Universal Robots PolyScope program: DAS428_958_02_MAR_21_DAS_lado_derecho.urp

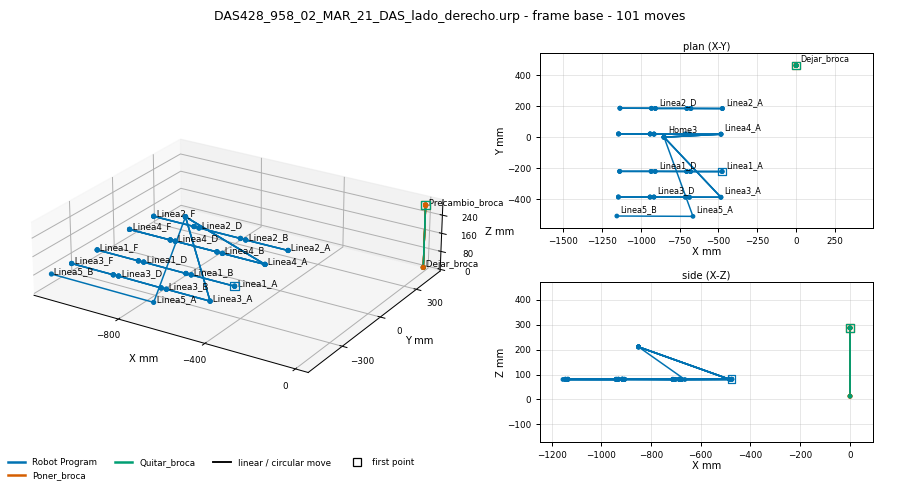
[picture p0: tool path of DAS428_958_02_MAR_21_DAS_lado_derecho.urp in frame base, 101 of 219 moves have a stored position in this frame; points joined in program order, loops and branches not executed]
Program DAS428_958_02_MAR_21_DAS_lado_derecho (installation=instalacion_26_FEB_21 directory=/programs/derecho createdIn=5.6.0.90886 lastSavedIn=5.6.0.90886 robotSerialNumber=20195001785)
Calibrated DH parameters: a=[0.000107, -0.568984, -0.552934, -0.00001, -0.000063, 0]; d=[0.180718, -257.998067, 200.685024, 57.48776, 0.119923, 0.115353]; alpha=[1.571119, 0.000876, -0.002498, 1.571178, -1.570523, 0]; deltaTheta=[0, -0.378191, 0.631587, -0.253396, 0, 0]
Robot Program (runOnlyOnce=false)
  Folder Variables
    bajada_broca := p[0,0,-0.008,0,0,0]
    barrenos_menos1 := 0
    barreno_actual := 0
    posicion := p[0,0,300,0,0,0]
    cambiar_broca := False
    barrenos_hechos := 0
    eje7 := 0
    Wait Sleep waitTime=0.5
  Folder Home
    Wait Sleep waitTime=0.3
    SafeHome (positionOptionType=SPEED_AND_ACCELERATION speed=1.047198 acceleration=1.396263 nextMotionTime=2)
    SuppressedNode
      MoveL speed 250 mm/s, acceleration 1200 mm/s^2 (useActiveTCP=true) feature=Base
        Waypoint home_trans: TCP in base x=-171.077 y=546.65 z=109.574 mm, rx=0.1544 ry=3.1247 rz=-0.2011 rad; joints [-91.802, -93.053, 127.954, -27.005, -275.278, -0.192] deg; TCP offset x=0.411 y=-218.298 z=37.994 mm, rx=1.558 ry=-0.1255 rz=0.1212 rad
    Wait Sleep waitTime=0.3
    iniciando_prog := True
    Call Poner_broca
  Folder Posicion2
    eje7 := 2
    Folder Broca_1
      Folder Linea1
        Folder Marcar_puntos
          MoveL speed 100 mm/s, acceleration 500 mm/s^2 (useActiveTCP=true) feature=Base
            SafeHome (positionOptionType=SPEED_AND_ACCELERATION speed=1.047198 acceleration=1.396263 nextMotionTime=2)
            Waypoint Linea1_A: TCP in base x=-476.23 y=-221.4 z=80.998 mm, rx=2.0263 ry=-2.3929 rz=-0.0208 rad; joints [8.239, -98.147, 138.323, -40.444, -261.448, -0.264] deg; TCP offset x=0.411 y=-218.298 z=37.994 mm, rx=1.558 ry=-0.1255 rz=0.1212 rad
            Waypoint Linea1_B: TCP in base x=-679.349 y=-221.301 z=80.412 mm, rx=2.0263 ry=-2.3929 rz=-0.0208 rad; joints [5.2, -80.225, 120.117, -40.154, -264.492, -0.236] deg
            Waypoint Linea1_C: TCP in base x=-704.534 y=-220.853 z=80.143 mm, rx=2.0263 ry=-2.3929 rz=-0.0208 rad; joints [4.927, -78.214, 117.618, -39.664, -264.765, -0.234] deg
            Waypoint Linea1_D: TCP in base x=-907.519 y=-220.332 z=80.645 mm, rx=2.0263 ry=-2.3929 rz=-0.0208 rad; joints [3.596, -62.527, 94.913, -32.645, -266.086, -0.228] deg
            Waypoint Linea1_E: TCP in base x=-933.182 y=-220.332 z=80.091 mm, rx=2.0263 ry=-2.3929 rz=-0.0208 rad; joints [3.48, -60.486, 91.71, -31.482, -266.199, -0.227] deg
            Waypoint Linea1_F: TCP in base x=-1136.071 y=-220.201 z=80.22 mm, rx=2.0263 ry=-2.3929 rz=-0.0208 rad; joints [2.763, -42.904, 61.27, -18.625, -266.887, -0.23] deg
        Folder AB
          'desbaste_inicial'
          bajada_broca := p[0,0,-0.008,0,0,0]
          barrenos_menos1 := 8
          barreno_actual := 0
          Loop While (checkContinuously=false) expression=barreno_actual≤barrenos_menos1
            Folder Perforacion
              MoveL speed 100 mm/s, acceleration 500 mm/s^2 (useActiveTCP=true) feature=Base
                internos := interpolate_pose(Linea1_A, Linea1_B, barreno_actual/barrenos_menos1)
                Waypoint Waypoint (Variable): variable=internos
                'desbaste_inicial'
                bajada_broca := p[0,0,-0.008,0,0,0]
                bajada := p[0,0,0.008,0,0,0]
                MoveDirectionNode (selectedDirection=ZMinus toolParams=0.003, 0.005)
                  Until DISTANCE (allowActions=false deceleration=3 distanceNodeType=STOP) Distance=0.045; motionParameters(blendRadius=0)
                Popup Message (haltProgram=false message=punto contacto alanzdo inputType=Text)
                MoveDirectionNode (selectedDirection=ZPlus toolParams=0.003, 0.005)
                  Until DISTANCE (allowActions=false deceleration=3 distanceNodeType=STOP) Distance=0.002; motionParameters(blendRadius=0)
                Wait Sleep waitTime=0.3
                Set DigitalOutput pin=config_out[1]; digitalValue=1
                Wait Sleep waitTime=0.3
                Loop Counting (count=3) loopVariable(name=Loop_11)
                  bajar := pose_add(get_actual_tcp_pose(), bajada_broca)
                  Waypoint Waypoint (Variable): motionParameters(jointSpeed=1.047198 jointAcceleration=1.396263 cartesianSpeed=0.001 cartesianAcceleration=0.005); variable=bajar
                  subir := pose_sub(get_actual_tcp_pose(), bajada_broca)
                  Waypoint Waypoint (Variable): motionParameters(jointSpeed=1.047198 jointAcceleration=1.396263 cartesianSpeed=0.005 cartesianAcceleration=0.01); variable=subir
                  bajada_broca := pose_sub(bajada_broca, bajada)
                MoveDirectionNode (selectedDirection=ZPlus toolParams=0.03, 0.035)
                  Until DISTANCE (allowActions=false deceleration=3 distanceNodeType=STOP) Distance=0.06; motionParameters(blendRadius=0)
                Set DigitalOutput pin=config_out[1]; digitalValue=0
                barreno_actual := barreno_actual+1
                Call Quitar_broca
                Call Poner_broca
        Folder CD
          'desbaste_inicial'
          bajada_broca := p[0,0,-0.008,0,0,0]
          barrenos_menos1 := 8
          barreno_actual := 0
          Loop While (checkContinuously=false) expression=barreno_actual≤barrenos_menos1
            Folder Perforacion
              MoveL speed 100 mm/s, acceleration 500 mm/s^2 (useActiveTCP=true) feature=Base
                internos := interpolate_pose(Linea1_C, Linea1_D, barreno_actual/barrenos_menos1)
                Waypoint Waypoint (Variable): variable=internos
                'desbaste_inicial'
                bajada_broca := p[0,0,-0.008,0,0,0]
                bajada := p[0,0,0.008,0,0,0]
                MoveDirectionNode (selectedDirection=ZMinus toolParams=0.003, 0.005)
                  Until DISTANCE (allowActions=false deceleration=3 distanceNodeType=STOP) Distance=0.045; motionParameters(blendRadius=0)
                Popup Message (haltProgram=false message=punto contacto alanzdo inputType=Text)
                MoveDirectionNode (selectedDirection=ZPlus toolParams=0.003, 0.005)
                  Until DISTANCE (allowActions=false deceleration=3 distanceNodeType=STOP) Distance=0.002; motionParameters(blendRadius=0)
                Wait Sleep waitTime=0.3
                Set DigitalOutput pin=config_out[1]; digitalValue=1
                Wait Sleep waitTime=0.3
                Loop Counting (count=3) loopVariable(name=Loop_14)
                  bajar := pose_add(get_actual_tcp_pose(), bajada_broca)
                  Waypoint Waypoint (Variable): motionParameters(jointSpeed=1.047198 jointAcceleration=1.396263 cartesianSpeed=0.001 cartesianAcceleration=0.005); variable=bajar
                  subir := pose_sub(get_actual_tcp_pose(), bajada_broca)
                  Waypoint Waypoint (Variable): motionParameters(jointSpeed=1.047198 jointAcceleration=1.396263 cartesianSpeed=0.005 cartesianAcceleration=0.01); variable=subir
                  bajada_broca := pose_sub(bajada_broca, bajada)
                MoveDirectionNode (selectedDirection=ZPlus toolParams=0.03, 0.035)
                  Until DISTANCE (allowActions=false deceleration=3 distanceNodeType=STOP) Distance=0.06; motionParameters(blendRadius=0)
                Set DigitalOutput pin=config_out[1]; digitalValue=0
                barreno_actual := barreno_actual+1
                Call Quitar_broca
                Call Poner_broca
        Folder EF
          'desbaste_inicial'
          bajada_broca := p[0,0,-0.008,0,0,0]
          barrenos_menos1 := 8
          barreno_actual := 0
          Loop While (checkContinuously=false) expression=barreno_actual≤barrenos_menos1
            Folder Perforacion
              MoveL speed 100 mm/s, acceleration 500 mm/s^2 (useActiveTCP=true) feature=Base
                internos := interpolate_pose(Linea1_E, Linea1_F, barreno_actual/barrenos_menos1)
                Waypoint Waypoint (Variable): variable=internos
                'desbaste_inicial'
                bajada_broca := p[0,0,-0.008,0,0,0]
                bajada := p[0,0,0.008,0,0,0]
                MoveDirectionNode (selectedDirection=ZMinus toolParams=0.003, 0.005)
                  Until DISTANCE (allowActions=false deceleration=3 distanceNodeType=STOP) Distance=0.045; motionParameters(blendRadius=0)
                Popup Message (haltProgram=false message=punto contacto alanzdo inputType=Text)
                MoveDirectionNode (selectedDirection=ZPlus toolParams=0.003, 0.005)
                  Until DISTANCE (allowActions=false deceleration=3 distanceNodeType=STOP) Distance=0.002; motionParameters(blendRadius=0)
                Wait Sleep waitTime=0.3
                Set DigitalOutput pin=config_out[1]; digitalValue=1
                Wait Sleep waitTime=0.3
                Loop Counting (count=3) loopVariable(name=Loop_16)
                  bajar := pose_add(get_actual_tcp_pose(), bajada_broca)
                  Waypoint Waypoint (Variable): motionParameters(jointSpeed=1.047198 jointAcceleration=1.396263 cartesianSpeed=0.001 cartesianAcceleration=0.005); variable=bajar
                  subir := pose_sub(get_actual_tcp_pose(), bajada_broca)
                  Waypoint Waypoint (Variable): motionParameters(jointSpeed=1.047198 jointAcceleration=1.396263 cartesianSpeed=0.005 cartesianAcceleration=0.01); variable=subir
                  bajada_broca := pose_sub(bajada_broca, bajada)
                MoveDirectionNode (selectedDirection=ZPlus toolParams=0.03, 0.035)
                  Until DISTANCE (allowActions=false deceleration=3 distanceNodeType=STOP) Distance=0.06; motionParameters(blendRadius=0)
                Set DigitalOutput pin=config_out[1]; digitalValue=0
                barreno_actual := barreno_actual+1
                Call Quitar_broca
                Call Poner_broca
      Popup Message (haltProgram=false message=Linea1 con chica Terminada! inputType=Text)
      Folder Linea2
        Folder Marcar_puntos
          MoveL speed 100 mm/s, acceleration 500 mm/s^2 (useActiveTCP=true) feature=Base
            Waypoint Linea2_A: TCP in base x=-474.583 y=184.454 z=81.011 mm, rx=2.0263 ry=-2.3928 rz=-0.0209 rad; joints [-57.964, -100.998, 140.513, -39.882, -327.65, 0.115] deg; TCP offset x=0.411 y=-218.298 z=37.994 mm, rx=1.558 ry=-0.1255 rz=0.1212 rad
            Waypoint Linea2_B: TCP in base x=-677.479 y=185.069 z=80.034 mm, rx=2.0263 ry=-2.3928 rz=-0.0209 rad; joints [-37.655, -81.603, 121.85, -40.529, -307.349, -0.029] deg
            Waypoint Linea2_C: TCP in base x=-703.112 y=185.207 z=80.706 mm, rx=2.0263 ry=-2.3928 rz=-0.0209 rad; joints [-36.031, -79.522, 119.204, -39.96, -305.725, -0.038] deg
            Waypoint Linea2_D: TCP in base x=-906.15 y=185.294 z=81.03 mm, rx=2.0263 ry=-2.3928 rz=-0.0209 rad; joints [-26.739, -63.46, 96.339, -33.14, -296.423, -0.088] deg
            Waypoint Linea2_E: TCP in base x=-931.212 y=185.988 z=81.375 mm, rx=2.0263 ry=-2.3928 rz=-0.0209 rad; joints [-25.954, -61.479, 93.157, -31.938, -295.635, -0.093] deg
            Waypoint Linea2_F: TCP in base x=-1134.161 y=186.61 z=81.262 mm, rx=2.0263 ry=-2.3928 rz=-0.0209 rad; joints [-20.753, -43.887, 62.952, -19.317, -290.406, -0.124] deg
        Folder AB
          'desbaste_inicial'
          bajada_broca := p[0,0,-0.008,0,0,0]
          barrenos_menos1 := 8
          barreno_actual := 0
          Loop While (checkContinuously=false) expression=barreno_actual≤barrenos_menos1
            Folder Perforacion
              MoveL speed 100 mm/s, acceleration 500 mm/s^2 (useActiveTCP=true) feature=Base
                internos := interpolate_pose(Linea2_A, Linea2_B, barreno_actual/barrenos_menos1)
                Waypoint Waypoint (Variable): variable=internos
                'desbaste_inicial'
                bajada_broca := p[0,0,-0.008,0,0,0]
                bajada := p[0,0,0.008,0,0,0]
                MoveDirectionNode (selectedDirection=ZMinus toolParams=0.003, 0.005)
                  Until DISTANCE (allowActions=false deceleration=3 distanceNodeType=STOP) Distance=0.045; motionParameters(blendRadius=0)
                Popup Message (haltProgram=false message=punto contacto alanzdo inputType=Text)
                MoveDirectionNode (selectedDirection=ZPlus toolParams=0.003, 0.005)
                  Until DISTANCE (allowActions=false deceleration=3 distanceNodeType=STOP) Distance=0.002; motionParameters(blendRadius=0)
                Wait Sleep waitTime=0.3
                Set DigitalOutput pin=config_out[1]; digitalValue=1
                Wait Sleep waitTime=0.3
                Loop Counting (count=3) loopVariable(name=Loop_2)
                  bajar := pose_add(get_actual_tcp_pose(), bajada_broca)
                  Waypoint Waypoint (Variable): motionParameters(jointSpeed=1.047198 jointAcceleration=1.396263 cartesianSpeed=0.001 cartesianAcceleration=0.005); variable=bajar
                  subir := pose_sub(get_actual_tcp_pose(), bajada_broca)
                  Waypoint Waypoint (Variable): motionParameters(jointSpeed=1.047198 jointAcceleration=1.396263 cartesianSpeed=0.005 cartesianAcceleration=0.01); variable=subir
                  bajada_broca := pose_sub(bajada_broca, bajada)
                MoveDirectionNode (selectedDirection=ZPlus toolParams=0.03, 0.035)
                  Until DISTANCE (allowActions=false deceleration=3 distanceNodeType=STOP) Distance=0.06; motionParameters(blendRadius=0)
                Set DigitalOutput pin=config_out[1]; digitalValue=0
                barreno_actual := barreno_actual+1
                Call Quitar_broca
                Call Poner_broca
        Folder CD
          'desbaste_inicial'
          bajada_broca := p[0,0,-0.008,0,0,0]
          barrenos_menos1 := 8
          barreno_actual := 0
          Loop While (checkContinuously=false) expression=barreno_actual≤barrenos_menos1
            Folder Perforacion
              MoveL speed 100 mm/s, acceleration 500 mm/s^2 (useActiveTCP=true) feature=Base
                internos := interpolate_pose(Linea2_C, Linea2_D, barreno_actual/barrenos_menos1)
                Waypoint Waypoint (Variable): variable=internos
                'desbaste_inicial'
                bajada_broca := p[0,0,-0.008,0,0,0]
                bajada := p[0,0,0.008,0,0,0]
                MoveDirectionNode (selectedDirection=ZMinus toolParams=0.003, 0.005)
                  Until DISTANCE (allowActions=false deceleration=3 distanceNodeType=STOP) Distance=0.045; motionParameters(blendRadius=0)
                Popup Message (haltProgram=false message=punto contacto alanzdo inputType=Text)
                MoveDirectionNode (selectedDirection=ZPlus toolParams=0.003, 0.005)
                  Until DISTANCE (allowActions=false deceleration=3 distanceNodeType=STOP) Distance=0.002; motionParameters(blendRadius=0)
                Wait Sleep waitTime=0.3
                Set DigitalOutput pin=config_out[1]; digitalValue=1
                Wait Sleep waitTime=0.3
                Loop Counting (count=3) loopVariable(name=Loop_5)
                  bajar := pose_add(get_actual_tcp_pose(), bajada_broca)
                  Waypoint Waypoint (Variable): motionParameters(jointSpeed=1.047198 jointAcceleration=1.396263 cartesianSpeed=0.001 cartesianAcceleration=0.005); variable=bajar
                  subir := pose_sub(get_actual_tcp_pose(), bajada_broca)
                  Waypoint Waypoint (Variable): motionParameters(jointSpeed=1.047198 jointAcceleration=1.396263 cartesianSpeed=0.005 cartesianAcceleration=0.01); variable=subir
                  bajada_broca := pose_sub(bajada_broca, bajada)
                MoveDirectionNode (selectedDirection=ZPlus toolParams=0.03, 0.035)
                  Until DISTANCE (allowActions=false deceleration=3 distanceNodeType=STOP) Distance=0.06; motionParameters(blendRadius=0)
                Set DigitalOutput pin=config_out[1]; digitalValue=0
                barreno_actual := barreno_actual+1
                Call Quitar_broca
                Call Poner_broca
        Folder EF
          'desbaste_inicial'
          bajada_broca := p[0,0,-0.008,0,0,0]
          barrenos_menos1 := 8
          barreno_actual := 0
          Loop While (checkContinuously=false) expression=barreno_actual≤barrenos_menos1
            Folder Perforacion
              MoveL speed 100 mm/s, acceleration 500 mm/s^2 (useActiveTCP=true) feature=Base
                internos := interpolate_pose(Linea2_E, Linea2_F, barreno_actual/barrenos_menos1)
                Waypoint Waypoint (Variable): variable=internos
                'desbaste_inicial'
                bajada_broca := p[0,0,-0.008,0,0,0]
                bajada := p[0,0,0.008,0,0,0]
                MoveDirectionNode (selectedDirection=ZMinus toolParams=0.003, 0.005)
                  Until DISTANCE (allowActions=false deceleration=3 distanceNodeType=STOP) Distance=0.045; motionParameters(blendRadius=0)
                Popup Message (haltProgram=false message=punto contacto alanzdo inputType=Text)
                MoveDirectionNode (selectedDirection=ZPlus toolParams=0.003, 0.005)
                  Until DISTANCE (allowActions=false deceleration=3 distanceNodeType=STOP) Distance=0.002; motionParameters(blendRadius=0)
                Wait Sleep waitTime=0.3
                Set DigitalOutput pin=config_out[1]; digitalValue=1
                Wait Sleep waitTime=0.3
                Loop Counting (count=3) loopVariable(name=Loop_9)
                  bajar := pose_add(get_actual_tcp_pose(), bajada_broca)
                  Waypoint Waypoint (Variable): motionParameters(jointSpeed=1.047198 jointAcceleration=1.396263 cartesianSpeed=0.001 cartesianAcceleration=0.005); variable=bajar
                  subir := pose_sub(get_actual_tcp_pose(), bajada_broca)
                  Waypoint Waypoint (Variable): motionParameters(jointSpeed=1.047198 jointAcceleration=1.396263 cartesianSpeed=0.005 cartesianAcceleration=0.01); variable=subir
                  bajada_broca := pose_sub(bajada_broca, bajada)
                MoveDirectionNode (selectedDirection=ZPlus toolParams=0.03, 0.035)
                  Until DISTANCE (allowActions=false deceleration=3 distanceNodeType=STOP) Distance=0.06; motionParameters(blendRadius=0)
                Set DigitalOutput pin=config_out[1]; digitalValue=0
                barreno_actual := barreno_actual+1
                If barreno_actual≥barrenos_menos1
                  cambiar_broca := True
                Call Quitar_broca
                Call Poner_broca
      Popup Message (haltProgram=false message=Linea2 con chica Terminada! inputType=Text)
    Folder Broca_2
      Folder Linea1
        Folder Marcar_puntos
          MoveL speed 100 mm/s, acceleration 500 mm/s^2 (useActiveTCP=true) feature=Base
            Waypoint Linea1_A: TCP in base x=-476.23 y=-221.4 z=80.998 mm, rx=2.0263 ry=-2.3929 rz=-0.0208 rad; joints [8.239, -98.147, 138.323, -40.444, -261.448, -0.264] deg; TCP offset x=0.411 y=-218.298 z=37.994 mm, rx=1.558 ry=-0.1255 rz=0.1212 rad
            Waypoint Linea1_B: TCP in base x=-679.349 y=-221.301 z=80.412 mm, rx=2.0263 ry=-2.3929 rz=-0.0208 rad; joints [5.2, -80.225, 120.117, -40.154, -264.492, -0.236] deg
            Waypoint Linea1_C: TCP in base x=-704.534 y=-220.853 z=80.143 mm, rx=2.0263 ry=-2.3929 rz=-0.0208 rad; joints [4.927, -78.214, 117.618, -39.664, -264.765, -0.234] deg
            Waypoint Linea1_D: TCP in base x=-907.519 y=-220.332 z=80.645 mm, rx=2.0263 ry=-2.3929 rz=-0.0208 rad; joints [3.596, -62.527, 94.913, -32.645, -266.086, -0.228] deg
            Waypoint Linea1_E: TCP in base x=-933.182 y=-220.332 z=80.091 mm, rx=2.0263 ry=-2.3929 rz=-0.0208 rad; joints [3.48, -60.486, 91.71, -31.482, -266.199, -0.227] deg
            Waypoint Linea1_F: TCP in base x=-1136.071 y=-220.201 z=80.22 mm, rx=2.0263 ry=-2.3929 rz=-0.0208 rad; joints [2.763, -42.904, 61.27, -18.625, -266.887, -0.23] deg
        Folder AB
          'desbaste_inicial'
          bajada_broca := p[0,0,-0.012,0,0,0]
          barrenos_menos1 := 8
          barreno_actual := 0
          Loop While (checkContinuously=false) expression=barreno_actual≤barrenos_menos1
            Folder Perforacion
              MoveL speed 100 mm/s, acceleration 500 mm/s^2 (useActiveTCP=true) feature=Base
                internos := interpolate_pose(Linea1_A, Linea1_B, barreno_actual/barrenos_menos1)
                Waypoint Waypoint (Variable): variable=internos
                'desbaste_inicial'
                bajada_broca := p[0,0,-0.012,0,0,0]
                bajada := p[0,0,0.012,0,0,0]
                MoveDirectionNode (selectedDirection=ZMinus toolParams=0.01, 0.015)
                  Until DISTANCE (allowActions=false deceleration=3 distanceNodeType=STOP) Distance=0.045; motionParameters(blendRadius=0)
                Popup Message (haltProgram=false message=punto contacto alanzdo inputType=Text)
                MoveDirectionNode (selectedDirection=ZPlus toolParams=0.003, 0.005)
                  Until DISTANCE (allowActions=false deceleration=3 distanceNodeType=STOP) Distance=0.001; motionParameters(blendRadius=0)
                Wait Sleep waitTime=0.3
                Set DigitalOutput pin=config_out[1]; digitalValue=1
                Wait Sleep waitTime=0.3
                Loop Counting (count=2) loopVariable(name=Loop_46)
                  bajar := pose_add(get_actual_tcp_pose(), bajada_broca)
                  Waypoint Waypoint (Variable): motionParameters(jointSpeed=1.047198 jointAcceleration=1.396263 cartesianSpeed=0.001 cartesianAcceleration=0.005); variable=bajar
                  subir := pose_sub(get_actual_tcp_pose(), bajada_broca)
                  Waypoint Waypoint (Variable): motionParameters(jointSpeed=1.047198 jointAcceleration=1.396263 cartesianSpeed=0.005 cartesianAcceleration=0.01); variable=subir
                  bajada_broca := pose_sub(bajada_broca, bajada)
                MoveDirectionNode (selectedDirection=ZPlus toolParams=0.03, 0.035)
                  Until DISTANCE (allowActions=false deceleration=3 distanceNodeType=STOP) Distance=0.06; motionParameters(blendRadius=0)
                Set DigitalOutput pin=config_out[1]; digitalValue=0
                barreno_actual := barreno_actual+1
                Call Quitar_broca
                Call Poner_broca
        Folder CD
          'desbaste_inicial'
          bajada_broca := p[0,0,-0.012,0,0,0]
          barrenos_menos1 := 8
          barreno_actual := 0
          Loop While (checkContinuously=false) expression=barreno_actual≤barrenos_menos1
            Folder Perforacion
              MoveL speed 100 mm/s, acceleration 500 mm/s^2 (useActiveTCP=true) feature=Base
                internos := interpolate_pose(Linea1_C, Linea1_D, barreno_actual/barrenos_menos1)
                Waypoint Waypoint (Variable): variable=internos
                'desbaste_inicial'
                bajada_broca := p[0,0,-0.012,0,0,0]
                bajada := p[0,0,0.012,0,0,0]
                MoveDirectionNode (selectedDirection=ZMinus toolParams=0.01, 0.015)
                  Until DISTANCE (allowActions=false deceleration=3 distanceNodeType=STOP) Distance=0.045; motionParameters(blendRadius=0)
                Popup Message (haltProgram=false message=punto contacto alanzdo inputType=Text)
                MoveDirectionNode (selectedDirection=ZPlus toolParams=0.003, 0.005)
                  Until DISTANCE (allowActions=false deceleration=3 distanceNodeType=STOP) Distance=0.001; motionParameters(blendRadius=0)
                Wait Sleep waitTime=0.3
                Set DigitalOutput pin=config_out[1]; digitalValue=1
                Wait Sleep waitTime=0.3
                Loop Counting (count=2) loopVariable(name=Loop_48)
                  bajar := pose_add(get_actual_tcp_pose(), bajada_broca)
                  Waypoint Waypoint (Variable): motionParameters(jointSpeed=1.047198 jointAcceleration=1.396263 cartesianSpeed=0.001 cartesianAcceleration=0.005); variable=bajar
                  subir := pose_sub(get_actual_tcp_pose(), bajada_broca)
                  Waypoint Waypoint (Variable): motionParameters(jointSpeed=1.047198 jointAcceleration=1.396263 cartesianSpeed=0.005 cartesianAcceleration=0.01); variable=subir
                  bajada_broca := pose_sub(bajada_broca, bajada)
                MoveDirectionNode (selectedDirection=ZPlus toolParams=0.03, 0.035)
                  Until DISTANCE (allowActions=false deceleration=3 distanceNodeType=STOP) Distance=0.06; motionParameters(blendRadius=0)
                Set DigitalOutput pin=config_out[1]; digitalValue=0
                barreno_actual := barreno_actual+1
                Call Quitar_broca
                Call Poner_broca
        Folder EF
          'desbaste_inicial'
          bajada_broca := p[0,0,-0.012,0,0,0]
          barrenos_menos1 := 8
          barreno_actual := 0
          Loop While (checkContinuously=false) expression=barreno_actual≤barrenos_menos1
            Folder Perforacion
              MoveL speed 100 mm/s, acceleration 500 mm/s^2 (useActiveTCP=true) feature=Base
                internos := interpolate_pose(Linea1_E, Linea1_F, barreno_actual/barrenos_menos1)
                Waypoint Waypoint (Variable): variable=internos
                'desbaste_inicial'
                bajada_broca := p[0,0,-0.012,0,0,0]
                bajada := p[0,0,0.012,0,0,0]
                MoveDirectionNode (selectedDirection=ZMinus toolParams=0.01, 0.015)
                  Until DISTANCE (allowActions=false deceleration=3 distanceNodeType=STOP) Distance=0.045; motionParameters(blendRadius=0)
                Popup Message (haltProgram=false message=punto contacto alanzdo inputType=Text)
                MoveDirectionNode (selectedDirection=ZPlus toolParams=0.003, 0.005)
                  Until DISTANCE (allowActions=false deceleration=3 distanceNodeType=STOP) Distance=0.001; motionParameters(blendRadius=0)
                Wait Sleep waitTime=0.3
                Set DigitalOutput pin=config_out[1]; digitalValue=1
                Wait Sleep waitTime=0.3
                Loop Counting (count=2) loopVariable(name=Loop_50)
                  bajar := pose_add(get_actual_tcp_pose(), bajada_broca)
                  Waypoint Waypoint (Variable): motionParameters(jointSpeed=1.047198 jointAcceleration=1.396263 cartesianSpeed=0.001 cartesianAcceleration=0.005); variable=bajar
                  subir := pose_sub(get_actual_tcp_pose(), bajada_broca)
                  Waypoint Waypoint (Variable): motionParameters(jointSpeed=1.047198 jointAcceleration=1.396263 cartesianSpeed=0.005 cartesianAcceleration=0.01); variable=subir
                  bajada_broca := pose_sub(bajada_broca, bajada)
                MoveDirectionNode (selectedDirection=ZPlus toolParams=0.03, 0.035)
                  Until DISTANCE (allowActions=false deceleration=3 distanceNodeType=STOP) Distance=0.06; motionParameters(blendRadius=0)
                Set DigitalOutput pin=config_out[1]; digitalValue=0
                barreno_actual := barreno_actual+1
                Call Quitar_broca
                Call Poner_broca
      Popup Message (haltProgram=false message=Linea1 con media Terminada! inputType=Text)
      Folder Linea2
        Folder Marcar_puntos
          MoveL speed 100 mm/s, acceleration 500 mm/s^2 (useActiveTCP=true) feature=Base
            Waypoint Linea2_A: TCP in base x=-474.583 y=184.454 z=81.011 mm, rx=2.0263 ry=-2.3928 rz=-0.0209 rad; joints [-57.964, -100.998, 140.513, -39.882, -327.65, 0.115] deg; TCP offset x=0.411 y=-218.298 z=37.994 mm, rx=1.558 ry=-0.1255 rz=0.1212 rad
            Waypoint Linea2_B: TCP in base x=-677.479 y=185.069 z=80.034 mm, rx=2.0263 ry=-2.3928 rz=-0.0209 rad; joints [-37.655, -81.603, 121.85, -40.529, -307.349, -0.029] deg
            Waypoint Linea2_C: TCP in base x=-703.112 y=185.207 z=80.706 mm, rx=2.0263 ry=-2.3928 rz=-0.0209 rad; joints [-36.031, -79.522, 119.204, -39.96, -305.725, -0.038] deg
            Waypoint Linea2_D: TCP in base x=-906.15 y=185.294 z=81.03 mm, rx=2.0263 ry=-2.3928 rz=-0.0209 rad; joints [-26.739, -63.46, 96.339, -33.14, -296.423, -0.088] deg
            Waypoint Linea2_E: TCP in base x=-931.212 y=185.988 z=81.375 mm, rx=2.0263 ry=-2.3928 rz=-0.0209 rad; joints [-25.954, -61.479, 93.157, -31.938, -295.635, -0.093] deg
            Waypoint Linea2_F: TCP in base x=-1134.161 y=186.61 z=81.262 mm, rx=2.0263 ry=-2.3928 rz=-0.0209 rad; joints [-20.753, -43.887, 62.952, -19.317, -290.406, -0.124] deg
        Folder AB
          'desbaste_inicial'
          bajada_broca := p[0,0,-0.012,0,0,0]
          barrenos_menos1 := 8
          barreno_actual := 0
          Loop While (checkContinuously=false) expression=barreno_actual≤barrenos_menos1
            Folder Perforacion
              MoveL speed 100 mm/s, acceleration 500 mm/s^2 (useActiveTCP=true) feature=Base
                internos := interpolate_pose(Linea2_A, Linea2_B, barreno_actual/barrenos_menos1)
                Waypoint Waypoint (Variable): variable=internos
                'desbaste_inicial'
                bajada_broca := p[0,0,-0.012,0,0,0]
                bajada := p[0,0,0.012,0,0,0]
                MoveDirectionNode (selectedDirection=ZMinus toolParams=0.003, 0.005)
                  Until DISTANCE (allowActions=false deceleration=3 distanceNodeType=STOP) Distance=0.045; motionParameters(blendRadius=0)
                Popup Message (haltProgram=false message=punto contacto alanzdo inputType=Text)
                MoveDirectionNode (selectedDirection=ZPlus toolParams=0.003, 0.005)
                  Until DISTANCE (allowActions=false deceleration=3 distanceNodeType=STOP) Distance=0.001; motionParameters(blendRadius=0)
                Wait Sleep waitTime=0.3
                Set DigitalOutput pin=config_out[1]; digitalValue=1
                Wait Sleep waitTime=0.3
                Loop Counting (count=2) loopVariable(name=Loop_34)
                  bajar := pose_add(get_actual_tcp_pose(), bajada_broca)
                  Waypoint Waypoint (Variable): motionParameters(jointSpeed=1.047198 jointAcceleration=1.396263 cartesianSpeed=0.001 cartesianAcceleration=0.005); variable=bajar
                  subir := pose_sub(get_actual_tcp_pose(), bajada_broca)
                  Waypoint Waypoint (Variable): motionParameters(jointSpeed=1.047198 jointAcceleration=1.396263 cartesianSpeed=0.005 cartesianAcceleration=0.01); variable=subir
                  bajada_broca := pose_sub(bajada_broca, bajada)
                MoveDirectionNode (selectedDirection=ZPlus toolParams=0.03, 0.035)
                  Until DISTANCE (allowActions=false deceleration=3 distanceNodeType=STOP) Distance=0.06; motionParameters(blendRadius=0)
                Set DigitalOutput pin=config_out[1]; digitalValue=0
                barreno_actual := barreno_actual+1
                Call Quitar_broca
                Call Poner_broca
        Folder CD
          'desbaste_inicial'
          bajada_broca := p[0,0,-0.012,0,0,0]
          barrenos_menos1 := 8
          barreno_actual := 0
          Loop While (checkContinuously=false) expression=barreno_actual≤barrenos_menos1
            Folder Perforacion
              MoveL speed 100 mm/s, acceleration 500 mm/s^2 (useActiveTCP=true) feature=Base
                internos := interpolate_pose(Linea2_C, Linea2_D, barreno_actual/barrenos_menos1)
                Waypoint Waypoint (Variable): variable=internos
                'desbaste_inicial'
                bajada_broca := p[0,0,-0.012,0,0,0]
                bajada := p[0,0,0.012,0,0,0]
                MoveDirectionNode (selectedDirection=ZMinus toolParams=0.003, 0.005)
                  Until DISTANCE (allowActions=false deceleration=3 distanceNodeType=STOP) Distance=0.045; motionParameters(blendRadius=0)
                Popup Message (haltProgram=false message=punto contacto alanzdo inputType=Text)
                MoveDirectionNode (selectedDirection=ZPlus toolParams=0.003, 0.005)
                  Until DISTANCE (allowActions=false deceleration=3 distanceNodeType=STOP) Distance=0.001; motionParameters(blendRadius=0)
                Wait Sleep waitTime=0.3
                Set DigitalOutput pin=config_out[1]; digitalValue=1
                Wait Sleep waitTime=0.3
                Loop Counting (count=2) loopVariable(name=Loop_36)
                  bajar := pose_add(get_actual_tcp_pose(), bajada_broca)
                  Waypoint Waypoint (Variable): motionParameters(jointSpeed=1.047198 jointAcceleration=1.396263 cartesianSpeed=0.001 cartesianAcceleration=0.005); variable=bajar
                  subir := pose_sub(get_actual_tcp_pose(), bajada_broca)
                  Waypoint Waypoint (Variable): motionParameters(jointSpeed=1.047198 jointAcceleration=1.396263 cartesianSpeed=0.005 cartesianAcceleration=0.01); variable=subir
                  bajada_broca := pose_sub(bajada_broca, bajada)
                MoveDirectionNode (selectedDirection=ZPlus toolParams=0.03, 0.035)
                  Until DISTANCE (allowActions=false deceleration=3 distanceNodeType=STOP) Distance=0.06; motionParameters(blendRadius=0)
                Set DigitalOutput pin=config_out[1]; digitalValue=0
                barreno_actual := barreno_actual+1
                Call Quitar_broca
                Call Poner_broca
        Folder EF
          'desbaste_inicial'
          bajada_broca := p[0,0,-0.012,0,0,0]
          barrenos_menos1 := 8
          barreno_actual := 0
          Loop While (checkContinuously=false) expression=barreno_actual≤barrenos_menos1
            Folder Perforacion
              MoveL speed 100 mm/s, acceleration 500 mm/s^2 (useActiveTCP=true) feature=Base
                internos := interpolate_pose(Linea2_E, Linea2_F, barreno_actual/barrenos_menos1)
                Waypoint Waypoint (Variable): variable=internos
                'desbaste_inicial'
                bajada_broca := p[0,0,-0.012,0,0,0]
                bajada := p[0,0,0.012,0,0,0]
                MoveDirectionNode (selectedDirection=ZMinus toolParams=0.003, 0.005)
                  Until DISTANCE (allowActions=false deceleration=3 distanceNodeType=STOP) Distance=0.045; motionParameters(blendRadius=0)
                Popup Message (haltProgram=false message=punto contacto alanzdo inputType=Text)
                MoveDirectionNode (selectedDirection=ZPlus toolParams=0.003, 0.005)
                  Until DISTANCE (allowActions=false deceleration=3 distanceNodeType=STOP) Distance=0.001; motionParameters(blendRadius=0)
                Wait Sleep waitTime=0.3
                Set DigitalOutput pin=config_out[1]; digitalValue=1
                Wait Sleep waitTime=0.3
                Loop Counting (count=2) loopVariable(name=Loop_38)
                  bajar := pose_add(get_actual_tcp_pose(), bajada_broca)
                  Waypoint Waypoint (Variable): motionParameters(jointSpeed=1.047198 jointAcceleration=1.396263 cartesianSpeed=0.001 cartesianAcceleration=0.005); variable=bajar
                  subir := pose_sub(get_actual_tcp_pose(), bajada_broca)
                  Waypoint Waypoint (Variable): motionParameters(jointSpeed=1.047198 jointAcceleration=1.396263 cartesianSpeed=0.005 cartesianAcceleration=0.01); variable=subir
                  bajada_broca := pose_sub(bajada_broca, bajada)
                MoveDirectionNode (selectedDirection=ZPlus toolParams=0.03, 0.035)
                  Until DISTANCE (allowActions=false deceleration=3 distanceNodeType=STOP) Distance=0.06; motionParameters(blendRadius=0)
                Set DigitalOutput pin=config_out[1]; digitalValue=0
                barreno_actual := barreno_actual+1
                If barreno_actual≥barrenos_menos1
                  cambiar_broca := True
                Call Quitar_broca
                Call Poner_broca
      Popup Message (haltProgram=false message=Linea2 con media Terminada! inputType=Text)
    Folder Broca_3
      Folder Linea1
        Folder Marcar_puntos
          MoveL speed 100 mm/s, acceleration 500 mm/s^2 (useActiveTCP=true) feature=Base
            Waypoint Linea1_A referenceName=Linea1_A: TCP in base x=-476.23 y=-221.4 z=80.998 mm, rx=2.0263 ry=-2.3929 rz=-0.0208 rad; joints [8.239, -98.147, 138.323, -40.444, -261.448, -0.264] deg; TCP offset x=0.411 y=-218.298 z=37.994 mm, rx=1.558 ry=-0.1255 rz=0.1212 rad
            Waypoint Linea1_B referenceName=Linea1_B: TCP in base x=-679.349 y=-221.301 z=80.412 mm, rx=2.0263 ry=-2.3929 rz=-0.0208 rad; joints [5.2, -80.225, 120.117, -40.154, -264.492, -0.236] deg
            Waypoint Linea1_C referenceName=Linea1_C: TCP in base x=-704.534 y=-220.853 z=80.143 mm, rx=2.0263 ry=-2.3929 rz=-0.0208 rad; joints [4.927, -78.214, 117.618, -39.664, -264.765, -0.234] deg
            Waypoint Linea1_D referenceName=Linea1_D: TCP in base x=-907.519 y=-220.332 z=80.645 mm, rx=2.0263 ry=-2.3929 rz=-0.0208 rad; joints [3.596, -62.527, 94.913, -32.645, -266.086, -0.228] deg
            Waypoint Linea1_E referenceName=Linea1_E: TCP in base x=-933.182 y=-220.332 z=80.091 mm, rx=2.0263 ry=-2.3929 rz=-0.0208 rad; joints [3.48, -60.486, 91.71, -31.482, -266.199, -0.227] deg
            Waypoint Linea1_F referenceName=Linea1_F: TCP in base x=-1136.071 y=-220.201 z=80.22 mm, rx=2.0263 ry=-2.3929 rz=-0.0208 rad; joints [2.763, -42.904, 61.27, -18.625, -266.887, -0.23] deg
        Folder AB
          'desbaste_inicial'
          bajada_broca := p[0,0,-0.012,0,0,0]
          barrenos_menos1 := 8
          barreno_actual := 0
          Loop While (checkContinuously=false) expression=barreno_actual≤barrenos_menos1
            Folder Perforacion
              MoveL speed 100 mm/s, acceleration 500 mm/s^2 (useActiveTCP=true) feature=Base
                internos := interpolate_pose(Linea1_A, Linea1_B, barreno_actual/barrenos_menos1)
                Waypoint Waypoint (Variable): variable=internos
                'desbaste_inicial'
                bajada_broca := p[0,0,-0.012,0,0,0]
                bajada := p[0,0,0.012,0,0,0]
                MoveDirectionNode (selectedDirection=ZMinus toolParams=0.01, 0.015)
                  Until DISTANCE (allowActions=false deceleration=3 distanceNodeType=STOP) Distance=0.045; motionParameters(blendRadius=0)
                Popup Message (haltProgram=false message=punto contacto alanzdo inputType=Text)
                MoveDirectionNode (selectedDirection=ZPlus toolParams=0.003, 0.005)
                  Until DISTANCE (allowActions=false deceleration=3 distanceNodeType=STOP) Distance=0.001; motionParameters(blendRadius=0)
                Wait Sleep waitTime=0.3
                Set DigitalOutput pin=config_out[1]; digitalValue=1
                Wait Sleep waitTime=0.3
                Loop Counting (count=2) loopVariable(name=Loop_18)
                  bajar := pose_add(get_actual_tcp_pose(), bajada_broca)
                  Waypoint Waypoint (Variable): motionParameters(jointSpeed=1.047198 jointAcceleration=1.396263 cartesianSpeed=0.001 cartesianAcceleration=0.005); variable=bajar
                  subir := pose_sub(get_actual_tcp_pose(), bajada_broca)
                  Waypoint Waypoint (Variable): motionParameters(jointSpeed=1.047198 jointAcceleration=1.396263 cartesianSpeed=0.005 cartesianAcceleration=0.01); variable=subir
                  bajada_broca := pose_sub(bajada_broca, bajada)
                MoveDirectionNode (selectedDirection=ZPlus toolParams=0.03, 0.035)
                  Until DISTANCE (allowActions=false deceleration=3 distanceNodeType=STOP) Distance=0.06; motionParameters(blendRadius=0)
                Set DigitalOutput pin=config_out[1]; digitalValue=0
                barreno_actual := barreno_actual+1
                Call Quitar_broca
                Call Poner_broca
        Folder CD
          'desbaste_inicial'
          bajada_broca := p[0,0,-0.012,0,0,0]
          barrenos_menos1 := 8
          barreno_actual := 0
          Loop While (checkContinuously=false) expression=barreno_actual≤barrenos_menos1
            Folder Perforacion
              MoveL speed 100 mm/s, acceleration 500 mm/s^2 (useActiveTCP=true) feature=Base
                internos := interpolate_pose(Linea1_C, Linea1_D, barreno_actual/barrenos_menos1)
                Waypoint Waypoint (Variable): variable=internos
                'desbaste_inicial'
                bajada_broca := p[0,0,-0.012,0,0,0]
                bajada := p[0,0,0.012,0,0,0]
                MoveDirectionNode (selectedDirection=ZMinus toolParams=0.01, 0.015)
                  Until DISTANCE (allowActions=false deceleration=3 distanceNodeType=STOP) Distance=0.045; motionParameters(blendRadius=0)
                Popup Message (haltProgram=false message=punto contacto alanzdo inputType=Text)
                MoveDirectionNode (selectedDirection=ZPlus toolParams=0.003, 0.005)
                  Until DISTANCE (allowActions=false deceleration=3 distanceNodeType=STOP) Distance=0.001; motionParameters(blendRadius=0)
                Wait Sleep waitTime=0.3
                Set DigitalOutput pin=config_out[1]; digitalValue=1
                Wait Sleep waitTime=0.3
                Loop Counting (count=2) loopVariable(name=Loop_20)
                  bajar := pose_add(get_actual_tcp_pose(), bajada_broca)
                  Waypoint Waypoint (Variable): motionParameters(jointSpeed=1.047198 jointAcceleration=1.396263 cartesianSpeed=0.001 cartesianAcceleration=0.005); variable=bajar
                  subir := pose_sub(get_actual_tcp_pose(), bajada_broca)
                  Waypoint Waypoint (Variable): motionParameters(jointSpeed=1.047198 jointAcceleration=1.396263 cartesianSpeed=0.005 cartesianAcceleration=0.01); variable=subir
                  bajada_broca := pose_sub(bajada_broca, bajada)
                MoveDirectionNode (selectedDirection=ZPlus toolParams=0.03, 0.035)
                  Until DISTANCE (allowActions=false deceleration=3 distanceNodeType=STOP) Distance=0.06; motionParameters(blendRadius=0)
                Set DigitalOutput pin=config_out[1]; digitalValue=0
                barreno_actual := barreno_actual+1
                Call Quitar_broca
                Call Poner_broca
        Folder EF
          'desbaste_inicial'
          bajada_broca := p[0,0,-0.012,0,0,0]
          barrenos_menos1 := 8
          barreno_actual := 0
          Loop While (checkContinuously=false) expression=barreno_actual≤barrenos_menos1
            Folder Perforacion
              MoveL speed 100 mm/s, acceleration 500 mm/s^2 (useActiveTCP=true) feature=Base
                internos := interpolate_pose(Linea1_E, Linea1_F, barreno_actual/barrenos_menos1)
                Waypoint Waypoint (Variable): variable=internos
                'desbaste_inicial'
                bajada_broca := p[0,0,-0.012,0,0,0]
                bajada := p[0,0,0.012,0,0,0]
                MoveDirectionNode (selectedDirection=ZMinus toolParams=0.01, 0.015)
                  Until DISTANCE (allowActions=false deceleration=3 distanceNodeType=STOP) Distance=0.045; motionParameters(blendRadius=0)
                Popup Message (haltProgram=false message=punto contacto alanzdo inputType=Text)
                MoveDirectionNode (selectedDirection=ZPlus toolParams=0.003, 0.005)
                  Until DISTANCE (allowActions=false deceleration=3 distanceNodeType=STOP) Distance=0.001; motionParameters(blendRadius=0)
                Wait Sleep waitTime=0.3
                Set DigitalOutput pin=config_out[1]; digitalValue=1
                Wait Sleep waitTime=0.3
                Loop Counting (count=2) loopVariable(name=Loop_22)
                  bajar := pose_add(get_actual_tcp_pose(), bajada_broca)
                  Waypoint Waypoint (Variable): motionParameters(jointSpeed=1.047198 jointAcceleration=1.396263 cartesianSpeed=0.001 cartesianAcceleration=0.005); variable=bajar
                  subir := pose_sub(get_actual_tcp_pose(), bajada_broca)
                  Waypoint Waypoint (Variable): motionParameters(jointSpeed=1.047198 jointAcceleration=1.396263 cartesianSpeed=0.005 cartesianAcceleration=0.01); variable=subir
                  bajada_broca := pose_sub(bajada_broca, bajada)
                MoveDirectionNode (selectedDirection=ZPlus toolParams=0.03, 0.035)
                  Until DISTANCE (allowActions=false deceleration=3 distanceNodeType=STOP) Distance=0.06; motionParameters(blendRadius=0)
                Set DigitalOutput pin=config_out[1]; digitalValue=0
                barreno_actual := barreno_actual+1
                Call Quitar_broca
                Call Poner_broca
      Popup Message (haltProgram=false message=Linea1 con full Terminada! inputType=Text)
      Folder Linea2
        Folder Marcar_puntos
          MoveL speed 100 mm/s, acceleration 500 mm/s^2 (useActiveTCP=true) feature=Base
            Waypoint Linea2_A: TCP in base x=-474.583 y=184.454 z=81.011 mm, rx=2.0263 ry=-2.3928 rz=-0.0209 rad; joints [-57.964, -100.998, 140.513, -39.882, -327.65, 0.115] deg; TCP offset x=0.411 y=-218.298 z=37.994 mm, rx=1.558 ry=-0.1255 rz=0.1212 rad
            Waypoint Linea2_B referenceName=Linea2_B: TCP in base x=-677.479 y=185.069 z=80.034 mm, rx=2.0263 ry=-2.3928 rz=-0.0209 rad; joints [-37.655, -81.603, 121.85, -40.529, -307.349, -0.029] deg
            Waypoint Linea2_C: TCP in base x=-703.112 y=185.207 z=80.706 mm, rx=2.0263 ry=-2.3928 rz=-0.0209 rad; joints [-36.031, -79.522, 119.204, -39.96, -305.725, -0.038] deg
            Waypoint Linea2_D: TCP in base x=-906.15 y=185.294 z=81.03 mm, rx=2.0263 ry=-2.3928 rz=-0.0209 rad; joints [-26.739, -63.46, 96.339, -33.14, -296.423, -0.088] deg
            Waypoint Linea2_E referenceName=Linea2_E: TCP in base x=-931.212 y=185.988 z=81.375 mm, rx=2.0263 ry=-2.3928 rz=-0.0209 rad; joints [-25.954, -61.479, 93.157, -31.938, -295.635, -0.093] deg
            Waypoint Linea2_F: TCP in base x=-1134.161 y=186.61 z=81.262 mm, rx=2.0263 ry=-2.3928 rz=-0.0209 rad; joints [-20.753, -43.887, 62.952, -19.317, -290.406, -0.124] deg
        Folder AB
          'desbaste_inicial'
          bajada_broca := p[0,0,-0.012,0,0,0]
          barrenos_menos1 := 8
          barreno_actual := 0
          Loop While (checkContinuously=false) expression=barreno_actual≤barrenos_menos1
            Folder Perforacion
              MoveL speed 100 mm/s, acceleration 500 mm/s^2 (useActiveTCP=true) feature=Base
                internos := interpolate_pose(Linea2_A, Linea2_B, barreno_actual/barrenos_menos1)
                Waypoint Waypoint (Variable): variable=internos
                'desbaste_inicial'
                bajada_broca := p[0,0,-0.012,0,0,0]
                bajada := p[0,0,0.012,0,0,0]
                MoveDirectionNode (selectedDirection=ZMinus toolParams=0.003, 0.005)
                  Until DISTANCE (allowActions=false deceleration=3 distanceNodeType=STOP) Distance=0.045; motionParameters(blendRadius=0)
                Popup Message (haltProgram=false message=punto contacto alanzdo inputType=Text)
                MoveDirectionNode (selectedDirection=ZPlus toolParams=0.003, 0.005)
                  Until DISTANCE (allowActions=false deceleration=3 distanceNodeType=STOP) Distance=0.001; motionParameters(blendRadius=0)
                Wait Sleep waitTime=0.3
                Set DigitalOutput pin=config_out[1]; digitalValue=1
                Wait Sleep waitTime=0.3
                Loop Counting (count=2) loopVariable(name=Loop_40)
                  bajar := pose_add(get_actual_tcp_pose(), bajada_broca)
                  Waypoint Waypoint (Variable): motionParameters(jointSpeed=1.047198 jointAcceleration=1.396263 cartesianSpeed=0.001 cartesianAcceleration=0.005); variable=bajar
                  subir := pose_sub(get_actual_tcp_pose(), bajada_broca)
                  Waypoint Waypoint (Variable): motionParameters(jointSpeed=1.047198 jointAcceleration=1.396263 cartesianSpeed=0.005 cartesianAcceleration=0.01); variable=subir
                  bajada_broca := pose_sub(bajada_broca, bajada)
                MoveDirectionNode (selectedDirection=ZPlus toolParams=0.03, 0.035)
                  Until DISTANCE (allowActions=false deceleration=3 distanceNodeType=STOP) Distance=0.06; motionParameters(blendRadius=0)
                Set DigitalOutput pin=config_out[1]; digitalValue=0
                barreno_actual := barreno_actual+1
                Call Quitar_broca
                Call Poner_broca
        Folder CD
          'desbaste_inicial'
          bajada_broca := p[0,0,-0.012,0,0,0]
          barrenos_menos1 := 8
          barreno_actual := 0
          Loop While (checkContinuously=false) expression=barreno_actual≤barrenos_menos1
            Folder Perforacion
              MoveL speed 100 mm/s, acceleration 500 mm/s^2 (useActiveTCP=true) feature=Base
                internos := interpolate_pose(Linea2_C, Linea2_D, barreno_actual/barrenos_menos1)
                Waypoint Waypoint (Variable): variable=internos
                'desbaste_inicial'
                bajada_broca := p[0,0,-0.012,0,0,0]
                bajada := p[0,0,0.012,0,0,0]
                MoveDirectionNode (selectedDirection=ZMinus toolParams=0.02, 0.025)
                  Until DISTANCE (allowActions=false deceleration=3 distanceNodeType=STOP) Distance=0.045; motionParameters(blendRadius=0)
                Popup Message (haltProgram=false message=punto contacto alanzdo inputType=Text)
                MoveDirectionNode (selectedDirection=ZPlus toolParams=0.003, 0.005)
                  Until DISTANCE (allowActions=false deceleration=3 distanceNodeType=STOP) Distance=0.001; motionParameters(blendRadius=0)
                Wait Sleep waitTime=0.3
                Set DigitalOutput pin=config_out[1]; digitalValue=1
                Wait Sleep waitTime=0.3
                Loop Counting (count=2) loopVariable(name=Loop_42)
                  bajar := pose_add(get_actual_tcp_pose(), bajada_broca)
                  Waypoint Waypoint (Variable): motionParameters(jointSpeed=1.047198 jointAcceleration=1.396263 cartesianSpeed=0.001 cartesianAcceleration=0.005); variable=bajar
                  subir := pose_sub(get_actual_tcp_pose(), bajada_broca)
                  Waypoint Waypoint (Variable): motionParameters(jointSpeed=1.047198 jointAcceleration=1.396263 cartesianSpeed=0.005 cartesianAcceleration=0.01); variable=subir
                  bajada_broca := pose_sub(bajada_broca, bajada)
                MoveDirectionNode (selectedDirection=ZPlus toolParams=0.03, 0.035)
                  Until DISTANCE (allowActions=false deceleration=3 distanceNodeType=STOP) Distance=0.06; motionParameters(blendRadius=0)
                Set DigitalOutput pin=config_out[1]; digitalValue=0
                barreno_actual := barreno_actual+1
                Call Quitar_broca
                Call Poner_broca
        Folder EF
          'desbaste_inicial'
          bajada_broca := p[0,0,-0.012,0,0,0]
          barrenos_menos1 := 8
          barreno_actual := 0
          Loop While (checkContinuously=false) expression=barreno_actual≤barrenos_menos1
            Folder Perforacion
              MoveL speed 100 mm/s, acceleration 500 mm/s^2 (useActiveTCP=true) feature=Base
                internos := interpolate_pose(Linea2_E, Linea2_F, barreno_actual/barrenos_menos1)
                Waypoint Waypoint (Variable): variable=internos
                'desbaste_inicial'
                bajada_broca := p[0,0,-0.012,0,0,0]
                bajada := p[0,0,0.012,0,0,0]
                MoveDirectionNode (selectedDirection=ZMinus toolParams=0.02, 0.025)
                  Until DISTANCE (allowActions=false deceleration=3 distanceNodeType=STOP) Distance=0.045; motionParameters(blendRadius=0)
                Popup Message (haltProgram=false message=punto contacto alanzdo inputType=Text)
                MoveDirectionNode (selectedDirection=ZPlus toolParams=0.003, 0.005)
                  Until DISTANCE (allowActions=false deceleration=3 distanceNodeType=STOP) Distance=0.001; motionParameters(blendRadius=0)
                Wait Sleep waitTime=0.3
                Set DigitalOutput pin=config_out[1]; digitalValue=1
                Wait Sleep waitTime=0.3
                Loop Counting (count=2) loopVariable(name=Loop_44)
                  bajar := pose_add(get_actual_tcp_pose(), bajada_broca)
                  Waypoint Waypoint (Variable): motionParameters(jointSpeed=1.047198 jointAcceleration=1.396263 cartesianSpeed=0.001 cartesianAcceleration=0.005); variable=bajar
                  subir := pose_sub(get_actual_tcp_pose(), bajada_broca)
                  Waypoint Waypoint (Variable): motionParameters(jointSpeed=1.047198 jointAcceleration=1.396263 cartesianSpeed=0.005 cartesianAcceleration=0.01); variable=subir
                  bajada_broca := pose_sub(bajada_broca, bajada)
                MoveDirectionNode (selectedDirection=ZPlus toolParams=0.03, 0.035)
                  Until DISTANCE (allowActions=false deceleration=3 distanceNodeType=STOP) Distance=0.06; motionParameters(blendRadius=0)
                Set DigitalOutput pin=config_out[1]; digitalValue=0
                barreno_actual := barreno_actual+1
                If barreno_actual≥barrenos_menos1
                  cambiar_broca := True
                Call Quitar_broca
                Call Poner_broca
      Popup Message (haltProgram=false message=Linea2 con full Terminada! inputType=Text)
  Folder Posicion3
    eje7 := 3
    Folder Broca_1
      Folder Linea3
        Folder Marcar_puntos
          MoveL speed 100 mm/s, acceleration 500 mm/s^2 (useActiveTCP=true) feature=Base
            Waypoint Home3: TCP in base x=-850.182 y=0 z=211.32 mm, rx=-2.0297 ry=2.3968 rz=0.0066 rad; joints [-14.374, -75.698, 98.757, -22.649, -284.037, -0.192] deg; TCP offset x=0.411 y=-218.298 z=37.994 mm, rx=1.558 ry=-0.1255 rz=0.1212 rad
            Waypoint Linea3_A: TCP in base x=-483.981 y=-387.033 z=81.05 mm, rx=-2.0297 ry=2.3968 rz=0.0065 rad; joints [29.472, -85.66, 126.185, -40.12, -240.222, 0.138] deg; TCP offset x=0.411 y=-218.298 z=37.994 mm, rx=1.558 ry=-0.1255 rz=0.1212 rad
            Waypoint Linea3_B: TCP in base x=-686.975 y=-386.566 z=81.205 mm, rx=-2.0297 ry=2.3968 rz=0.0065 rad; joints [20.619, -72.662, 109.808, -36.76, -249.072, 0.076] deg
            Waypoint Linea3_C: TCP in base x=-712.354 y=-386.033 z=80.584 mm, rx=-2.0297 ry=2.3968 rz=0.0065 rad; joints [19.8, -70.954, 107.463, -36.125, -249.889, 0.07] deg
            Waypoint Linea3_D: TCP in base x=-915.146 y=-385.55 z=81.731 mm, rx=-2.0297 ry=2.3968 rz=0.0065 rad; joints [15.111, -56.737, 85.163, -28.047, -254.563, 0.035] deg
            Waypoint Linea3_E: TCP in base x=-940.448 y=-385.682 z=81.142 mm, rx=-2.0297 ry=2.3968 rz=0.0065 rad; joints [14.681, -54.779, 81.937, -26.78, -254.99, 0.031] deg
            Waypoint Linea3_F: TCP in base x=-1144.267 y=-385.383 z=81.233 mm, rx=-2.0297 ry=2.3968 rz=0.0065 rad; joints [11.857, -36.303, 48.734, -12.056, -257.778, 0.006] deg
        Folder AB
          'desbaste_inicial'
          bajada_broca := p[0,0,-0.008,0,0,0]
          barrenos_menos1 := 8
          barreno_actual := 0
          Loop While (checkContinuously=false) expression=barreno_actual≤barrenos_menos1
            Folder Perforacion
              MoveL speed 100 mm/s, acceleration 500 mm/s^2 (useActiveTCP=true) feature=Base
                internos := interpolate_pose(Linea3_A, Linea3_B, barreno_actual/barrenos_menos1)
                Waypoint Waypoint (Variable): variable=internos
                'desbaste_inicial'
                bajada_broca := p[0,0,-0.008,0,0,0]
                bajada := p[0,0,0.008,0,0,0]
                MoveDirectionNode (selectedDirection=ZMinus toolParams=0.02, 0.015)
                  Until DISTANCE (allowActions=false deceleration=3 distanceNodeType=STOP) Distance=0.055; motionParameters(blendRadius=0)
                Popup Message (haltProgram=false message=punto contacto alanzdo inputType=Text)
                MoveDirectionNode (selectedDirection=ZPlus toolParams=0.003, 0.005)
                  Until DISTANCE (allowActions=false deceleration=3 distanceNodeType=STOP) Distance=0.002; motionParameters(blendRadius=0)
                Wait Sleep waitTime=0.3
                Set DigitalOutput pin=config_out[1]; digitalValue=1
                Wait Sleep waitTime=0.3
                Loop Counting (count=3) loopVariable(name=Loop_3)
                  bajar := pose_add(get_actual_tcp_pose(), bajada_broca)
                  Waypoint Waypoint (Variable): motionParameters(jointSpeed=1.047198 jointAcceleration=1.396263 cartesianSpeed=0.001 cartesianAcceleration=0.005); variable=bajar
                  subir := pose_sub(get_actual_tcp_pose(), bajada_broca)
                  Waypoint Waypoint (Variable): motionParameters(jointSpeed=1.047198 jointAcceleration=1.396263 cartesianSpeed=0.01 cartesianAcceleration=0.01); variable=subir
                  bajada_broca := pose_sub(bajada_broca, bajada)
                MoveDirectionNode (selectedDirection=ZPlus toolParams=0.03, 0.035)
                  Until DISTANCE (allowActions=false deceleration=3 distanceNodeType=STOP) Distance=0.06; motionParameters(blendRadius=0)
                Set DigitalOutput pin=config_out[1]; digitalValue=0
                barreno_actual := barreno_actual+1
                SuppressedNode
                  Call Quitar_broca
                SuppressedNode
                  Call Poner_broca
        Folder CD
          'desbaste_inicial'
          bajada_broca := p[0,0,-0.008,0,0,0]
          barrenos_menos1 := 8
          barreno_actual := 0
          Loop While (checkContinuously=false) expression=barreno_actual≤barrenos_menos1
            Folder Perforacion
              MoveL speed 100 mm/s, acceleration 500 mm/s^2 (useActiveTCP=true) feature=Base
                internos := interpolate_pose(Linea3_C, Linea3_D, barreno_actual/barrenos_menos1)
                Waypoint Waypoint (Variable): variable=internos
                'desbaste_inicial'
                bajada_broca := p[0,0,-0.008,0,0,0]
                bajada := p[0,0,0.008,0,0,0]
                MoveDirectionNode (selectedDirection=ZMinus toolParams=0.02, 0.015)
                  Until DISTANCE (allowActions=false deceleration=3 distanceNodeType=STOP) Distance=0.055; motionParameters(blendRadius=0)
                Popup Message (haltProgram=false message=punto contacto alanzdo inputType=Text)
                MoveDirectionNode (selectedDirection=ZPlus toolParams=0.003, 0.005)
                  Until DISTANCE (allowActions=false deceleration=3 distanceNodeType=STOP) Distance=0.002; motionParameters(blendRadius=0)
                Wait Sleep waitTime=0.3
                Set DigitalOutput pin=config_out[1]; digitalValue=1
                Wait Sleep waitTime=0.3
                Loop Counting (count=3) loopVariable(name=Loop_6)
                  bajar := pose_add(get_actual_tcp_pose(), bajada_broca)
                  Waypoint Waypoint (Variable): motionParameters(jointSpeed=1.047198 jointAcceleration=1.396263 cartesianSpeed=0.001 cartesianAcceleration=0.005); variable=bajar
                  subir := pose_sub(get_actual_tcp_pose(), bajada_broca)
                  Waypoint Waypoint (Variable): motionParameters(jointSpeed=1.047198 jointAcceleration=1.396263 cartesianSpeed=0.01 cartesianAcceleration=0.01); variable=subir
                  bajada_broca := pose_sub(bajada_broca, bajada)
                MoveDirectionNode (selectedDirection=ZPlus toolParams=0.03, 0.035)
                  Until DISTANCE (allowActions=false deceleration=3 distanceNodeType=STOP) Distance=0.06; motionParameters(blendRadius=0)
                Set DigitalOutput pin=config_out[1]; digitalValue=0
                barreno_actual := barreno_actual+1
                SuppressedNode
                  Call Quitar_broca
                SuppressedNode
                  Call Poner_broca
        Folder EF
          'desbaste_inicial'
          bajada_broca := p[0,0,-0.008,0,0,0]
          barrenos_menos1 := 8
          barreno_actual := 0
          Loop While (checkContinuously=false) expression=barreno_actual≤barrenos_menos1
            Folder Perforacion
              MoveL speed 100 mm/s, acceleration 500 mm/s^2 (useActiveTCP=true) feature=Base
                internos := interpolate_pose(Linea3_E, Linea3_F, barreno_actual/barrenos_menos1)
                Waypoint Waypoint (Variable): variable=internos
                'desbaste_inicial'
                bajada_broca := p[0,0,-0.008,0,0,0]
                bajada := p[0,0,0.008,0,0,0]
                MoveDirectionNode (selectedDirection=ZMinus toolParams=0.02, 0.015)
                  Until DISTANCE (allowActions=false deceleration=3 distanceNodeType=STOP) Distance=0.055; motionParameters(blendRadius=0)
                Popup Message (haltProgram=false message=punto contacto alanzdo inputType=Text)
                MoveDirectionNode (selectedDirection=ZPlus toolParams=0.003, 0.005)
                  Until DISTANCE (allowActions=false deceleration=3 distanceNodeType=STOP) Distance=0.002; motionParameters(blendRadius=0)
                Wait Sleep waitTime=0.3
                Set DigitalOutput pin=config_out[1]; digitalValue=1
                Wait Sleep waitTime=0.3
                Loop Counting (count=3) loopVariable(name=Loop_8)
                  bajar := pose_add(get_actual_tcp_pose(), bajada_broca)
                  Waypoint Waypoint (Variable): motionParameters(jointSpeed=1.047198 jointAcceleration=1.396263 cartesianSpeed=0.001 cartesianAcceleration=0.005); variable=bajar
                  subir := pose_sub(get_actual_tcp_pose(), bajada_broca)
                  Waypoint Waypoint (Variable): motionParameters(jointSpeed=1.047198 jointAcceleration=1.396263 cartesianSpeed=0.01 cartesianAcceleration=0.01); variable=subir
                  bajada_broca := pose_sub(bajada_broca, bajada)
                MoveDirectionNode (selectedDirection=ZPlus toolParams=0.03, 0.035)
                  Until DISTANCE (allowActions=false deceleration=3 distanceNodeType=STOP) Distance=0.06; motionParameters(blendRadius=0)
                Set DigitalOutput pin=config_out[1]; digitalValue=0
                barreno_actual := barreno_actual+1
                SuppressedNode
                  Call Quitar_broca
                SuppressedNode
                  Call Poner_broca
      Popup Message (haltProgram=false message=Linea3 con chica Terminada! inputType=Text)
      Folder Linea4
        Folder Marcar_puntos
          MoveL speed 100 mm/s, acceleration 500 mm/s^2 (useActiveTCP=true) feature=Base
            Waypoint Home3: TCP in base x=-850.182 y=0 z=211.32 mm, rx=-2.0297 ry=2.3968 rz=0.0066 rad; joints [-14.374, -75.698, 98.757, -22.649, -284.037, -0.192] deg; TCP offset x=0.411 y=-218.298 z=37.994 mm, rx=1.558 ry=-0.1255 rz=0.1212 rad
            Waypoint Linea4_A: TCP in base x=-483.35 y=19.133 z=80.413 mm, rx=-2.0297 ry=2.3968 rz=0.0066 rad; joints [-34.857, -105.949, 143.743, -37.281, -304.535, -0.37] deg
            Waypoint Linea4_B: TCP in base x=-685.405 y=19.216 z=80.605 mm, rx=-2.0297 ry=2.3968 rz=0.0066 rad; joints [-21.02, -83.488, 123.782, -39.869, -290.712, -0.217] deg
            Waypoint Linea4_C: TCP in base x=-711.768 y=19.56 z=80.904 mm, rx=-2.0297 ry=2.3968 rz=0.0066 rad; joints [-20.032, -81.151, 120.968, -39.396, -289.723, -0.208] deg
            Waypoint Linea4_D: TCP in base x=-914.58 y=19.801 z=80.703 mm, rx=-2.0297 ry=2.3968 rz=0.0066 rad; joints [-14.612, -64.317, 97.516, -32.795, -284.295, -0.166] deg
            Waypoint Linea4_E: TCP in base x=-939.799 y=20.701 z=80.126 mm, rx=-2.0297 ry=2.3968 rz=0.0066 rad; joints [-14.202, -62.236, 94.311, -31.673, -283.882, -0.163] deg
            Waypoint Linea4_F: TCP in base x=-1143.008 y=20.924 z=80.361 mm, rx=-2.0297 ry=2.3968 rz=0.0066 rad; joints [-11.271, -44.369, 63.742, -18.977, -280.923, -0.147] deg
        Folder AB
          'desbaste_inicial'
          bajada_broca := p[0,0,-0.008,0,0,0]
          barrenos_menos1 := 8
          barreno_actual := 0
          Loop While (checkContinuously=false) expression=barreno_actual≤barrenos_menos1
            Folder Perforacion
              MoveL speed 100 mm/s, acceleration 500 mm/s^2 (useActiveTCP=true) feature=Base
                internos := interpolate_pose(Linea4_A, Linea4_B, barreno_actual/barrenos_menos1)
                Waypoint Waypoint (Variable): variable=internos
                'desbaste_inicial'
                bajada_broca := p[0,0,-0.008,0,0,0]
                bajada := p[0,0,0.008,0,0,0]
                MoveDirectionNode (selectedDirection=ZMinus toolParams=0.02, 0.015)
                  Until DISTANCE (allowActions=false deceleration=3 distanceNodeType=STOP) Distance=0.055; motionParameters(blendRadius=0)
                Popup Message (haltProgram=false message=punto contacto alanzdo inputType=Text)
                MoveDirectionNode (selectedDirection=ZPlus toolParams=0.003, 0.005)
                  Until DISTANCE (allowActions=false deceleration=3 distanceNodeType=STOP) Distance=0.002; motionParameters(blendRadius=0)
                Wait Sleep waitTime=0.3
                Set DigitalOutput pin=config_out[1]; digitalValue=1
                Wait Sleep waitTime=0.3
                Loop Counting (count=3) loopVariable(name=Loop_12)
                  bajar := pose_add(get_actual_tcp_pose(), bajada_broca)
                  Waypoint Waypoint (Variable): motionParameters(jointSpeed=1.047198 jointAcceleration=1.396263 cartesianSpeed=0.001 cartesianAcceleration=0.005); variable=bajar
                  subir := pose_sub(get_actual_tcp_pose(), bajada_broca)
                  Waypoint Waypoint (Variable): motionParameters(jointSpeed=1.047198 jointAcceleration=1.396263 cartesianSpeed=0.01 cartesianAcceleration=0.01); variable=subir
                  bajada_broca := pose_sub(bajada_broca, bajada)
                MoveDirectionNode (selectedDirection=ZPlus toolParams=0.03, 0.035)
                  Until DISTANCE (allowActions=false deceleration=3 distanceNodeType=STOP) Distance=0.06; motionParameters(blendRadius=0)
                Set DigitalOutput pin=config_out[1]; digitalValue=0
                barreno_actual := barreno_actual+1
                SuppressedNode
                  Call Quitar_broca
                SuppressedNode
                  Call Poner_broca
        Folder CD
          'desbaste_inicial'
          bajada_broca := p[0,0,-0.008,0,0,0]
          barrenos_menos1 := 8
          barreno_actual := 0
          Loop While (checkContinuously=false) expression=barreno_actual≤barrenos_menos1
            Folder Perforacion
              MoveL speed 100 mm/s, acceleration 500 mm/s^2 (useActiveTCP=true) feature=Base
                internos := interpolate_pose(Linea4_C, Linea4_D, barreno_actual/barrenos_menos1)
                Waypoint Waypoint (Variable): variable=internos
                'desbaste_inicial'
                bajada_broca := p[0,0,-0.008,0,0,0]
                bajada := p[0,0,0.008,0,0,0]
                MoveDirectionNode (selectedDirection=ZMinus toolParams=0.02, 0.015)
                  Until DISTANCE (allowActions=false deceleration=3 distanceNodeType=STOP) Distance=0.055; motionParameters(blendRadius=0)
                Popup Message (haltProgram=false message=punto contacto alanzdo inputType=Text)
                MoveDirectionNode (selectedDirection=ZPlus toolParams=0.003, 0.005)
                  Until DISTANCE (allowActions=false deceleration=3 distanceNodeType=STOP) Distance=0.002; motionParameters(blendRadius=0)
                Wait Sleep waitTime=0.3
                Set DigitalOutput pin=config_out[1]; digitalValue=1
                Wait Sleep waitTime=0.3
                Loop Counting (count=3) loopVariable(name=Loop_15)
                  bajar := pose_add(get_actual_tcp_pose(), bajada_broca)
                  Waypoint Waypoint (Variable): motionParameters(jointSpeed=1.047198 jointAcceleration=1.396263 cartesianSpeed=0.001 cartesianAcceleration=0.005); variable=bajar
                  subir := pose_sub(get_actual_tcp_pose(), bajada_broca)
                  Waypoint Waypoint (Variable): motionParameters(jointSpeed=1.047198 jointAcceleration=1.396263 cartesianSpeed=0.01 cartesianAcceleration=0.01); variable=subir
                  bajada_broca := pose_sub(bajada_broca, bajada)
                MoveDirectionNode (selectedDirection=ZPlus toolParams=0.03, 0.035)
                  Until DISTANCE (allowActions=false deceleration=3 distanceNodeType=STOP) Distance=0.06; motionParameters(blendRadius=0)
                Set DigitalOutput pin=config_out[1]; digitalValue=0
                barreno_actual := barreno_actual+1
                SuppressedNode
                  Call Quitar_broca
                SuppressedNode
                  Call Poner_broca
        Folder EF
          'desbaste_inicial'
          bajada_broca := p[0,0,-0.008,0,0,0]
          barrenos_menos1 := 8
          barreno_actual := 0
          Loop While (checkContinuously=false) expression=barreno_actual≤barrenos_menos1
            Folder Perforacion
              MoveL speed 100 mm/s, acceleration 500 mm/s^2 (useActiveTCP=true) feature=Base
                internos := interpolate_pose(Linea4_E, Linea4_F, barreno_actual/barrenos_menos1)
                Waypoint Waypoint (Variable): variable=internos
                'desbaste_inicial'
                bajada_broca := p[0,0,-0.008,0,0,0]
                bajada := p[0,0,0.008,0,0,0]
                MoveDirectionNode (selectedDirection=ZMinus toolParams=0.02, 0.015)
                  Until DISTANCE (allowActions=false deceleration=3 distanceNodeType=STOP) Distance=0.055; motionParameters(blendRadius=0)
                Popup Message (haltProgram=false message=punto contacto alanzdo inputType=Text)
                MoveDirectionNode (selectedDirection=ZPlus toolParams=0.003, 0.005)
                  Until DISTANCE (allowActions=false deceleration=3 distanceNodeType=STOP) Distance=0.002; motionParameters(blendRadius=0)
                Wait Sleep waitTime=0.3
                Set DigitalOutput pin=config_out[1]; digitalValue=1
                Wait Sleep waitTime=0.3
                Loop Counting (count=3) loopVariable(name=Loop_19)
                  bajar := pose_add(get_actual_tcp_pose(), bajada_broca)
                  Waypoint Waypoint (Variable): motionParameters(jointSpeed=1.047198 jointAcceleration=1.396263 cartesianSpeed=0.001 cartesianAcceleration=0.005); variable=bajar
                  subir := pose_sub(get_actual_tcp_pose(), bajada_broca)
                  Waypoint Waypoint (Variable): motionParameters(jointSpeed=1.047198 jointAcceleration=1.396263 cartesianSpeed=0.01 cartesianAcceleration=0.01); variable=subir
                  bajada_broca := pose_sub(bajada_broca, bajada)
                MoveDirectionNode (selectedDirection=ZPlus toolParams=0.03, 0.035)
                  Until DISTANCE (allowActions=false deceleration=3 distanceNodeType=STOP) Distance=0.06; motionParameters(blendRadius=0)
                Set DigitalOutput pin=config_out[1]; digitalValue=0
                barreno_actual := barreno_actual+1
                If barreno_actual≥barrenos_menos1
                  cambiar_broca := True
                SuppressedNode
                  Call Quitar_broca
                SuppressedNode
                  Call Poner_broca
      Popup Message (haltProgram=false message=Linea4 con chica Terminada! inputType=Text)
    Folder Broca_2
      Folder Linea3
        Folder Marcar_puntos
          MoveL speed 100 mm/s, acceleration 500 mm/s^2 (useActiveTCP=true) feature=Base
            Waypoint Home3: TCP in base x=-850.182 y=0 z=211.32 mm, rx=-2.0297 ry=2.3968 rz=0.0066 rad; joints [-14.374, -75.698, 98.757, -22.649, -284.037, -0.192] deg
            Waypoint Linea3_A: TCP in base x=-483.981 y=-387.033 z=81.05 mm, rx=-2.0297 ry=2.3968 rz=0.0065 rad; joints [29.472, -85.66, 126.185, -40.12, -240.222, 0.138] deg; TCP offset x=0.411 y=-218.298 z=37.994 mm, rx=1.558 ry=-0.1255 rz=0.1212 rad
            Waypoint Linea3_B: TCP in base x=-686.975 y=-386.566 z=81.205 mm, rx=-2.0297 ry=2.3968 rz=0.0065 rad; joints [20.619, -72.662, 109.808, -36.76, -249.072, 0.076] deg
            Waypoint Linea3_C: TCP in base x=-712.354 y=-386.033 z=80.584 mm, rx=-2.0297 ry=2.3968 rz=0.0065 rad; joints [19.8, -70.954, 107.463, -36.125, -249.889, 0.07] deg
            Waypoint Linea3_D: TCP in base x=-915.146 y=-385.55 z=81.731 mm, rx=-2.0297 ry=2.3968 rz=0.0065 rad; joints [15.111, -56.737, 85.163, -28.047, -254.563, 0.035] deg
            Waypoint Linea3_E: TCP in base x=-940.448 y=-385.682 z=81.142 mm, rx=-2.0297 ry=2.3968 rz=0.0065 rad; joints [14.681, -54.779, 81.937, -26.78, -254.99, 0.031] deg
            Waypoint Linea3_F: TCP in base x=-1144.267 y=-385.383 z=81.233 mm, rx=-2.0297 ry=2.3968 rz=0.0065 rad; joints [11.857, -36.303, 48.734, -12.056, -257.778, 0.006] deg
        Folder AB
          'desbaste_inicial'
          bajada_broca := p[0,0,-0.012,0,0,0]
          barrenos_menos1 := 8
          barreno_actual := 0
          Loop While (checkContinuously=false) expression=barreno_actual≤barrenos_menos1
            Folder Perforacion
              MoveL speed 100 mm/s, acceleration 500 mm/s^2 (useActiveTCP=true) feature=Base
                internos := interpolate_pose(Linea3_A, Linea3_B, barreno_actual/barrenos_menos1)
                Waypoint Waypoint (Variable): variable=internos
                'desbaste_inicial'
                bajada_broca := p[0,0,-0.012,0,0,0]
                bajada := p[0,0,0.012,0,0,0]
                MoveDirectionNode (selectedDirection=ZMinus toolParams=0.02, 0.015)
                  Until DISTANCE (allowActions=false deceleration=3 distanceNodeType=STOP) Distance=0.055; motionParameters(blendRadius=0)
                Popup Message (haltProgram=false message=punto contacto alanzdo inputType=Text)
                MoveDirectionNode (selectedDirection=ZPlus toolParams=0.003, 0.005)
                  Until DISTANCE (allowActions=false deceleration=3 distanceNodeType=STOP) Distance=0.001; motionParameters(blendRadius=0)
                Wait Sleep waitTime=0.3
                Set DigitalOutput pin=config_out[1]; digitalValue=1
                Wait Sleep waitTime=0.3
                Loop Counting (count=2) loopVariable(name=Loop_23)
                  bajar := pose_add(get_actual_tcp_pose(), bajada_broca)
                  Waypoint Waypoint (Variable): motionParameters(jointSpeed=1.047198 jointAcceleration=1.396263 cartesianSpeed=0.001 cartesianAcceleration=0.005); variable=bajar
                  subir := pose_sub(get_actual_tcp_pose(), bajada_broca)
                  Waypoint Waypoint (Variable): motionParameters(jointSpeed=1.047198 jointAcceleration=1.396263 cartesianSpeed=0.01 cartesianAcceleration=0.01); variable=subir
                  bajada_broca := pose_sub(bajada_broca, bajada)
                MoveDirectionNode (selectedDirection=ZPlus toolParams=0.03, 0.035)
                  Until DISTANCE (allowActions=false deceleration=3 distanceNodeType=STOP) Distance=0.06; motionParameters(blendRadius=0)
                Set DigitalOutput pin=config_out[1]; digitalValue=0
                barreno_actual := barreno_actual+1
                SuppressedNode
                  Call Quitar_broca
                SuppressedNode
                  Call Poner_broca
        Folder CD
          'desbaste_inicial'
          bajada_broca := p[0,0,-0.012,0,0,0]
          barrenos_menos1 := 8
          barreno_actual := 0
          Loop While (checkContinuously=false) expression=barreno_actual≤barrenos_menos1
            Folder Perforacion
              MoveL speed 100 mm/s, acceleration 500 mm/s^2 (useActiveTCP=true) feature=Base
                internos := interpolate_pose(Linea3_C, Linea3_D, barreno_actual/barrenos_menos1)
                Waypoint Waypoint (Variable): variable=internos
                'desbaste_inicial'
                bajada_broca := p[0,0,-0.012,0,0,0]
                bajada := p[0,0,0.012,0,0,0]
                MoveDirectionNode (selectedDirection=ZMinus toolParams=0.02, 0.015)
                  Until DISTANCE (allowActions=false deceleration=3 distanceNodeType=STOP) Distance=0.055; motionParameters(blendRadius=0)
                Popup Message (haltProgram=false message=punto contacto alanzdo inputType=Text)
                MoveDirectionNode (selectedDirection=ZPlus toolParams=0.003, 0.005)
                  Until DISTANCE (allowActions=false deceleration=3 distanceNodeType=STOP) Distance=0.001; motionParameters(blendRadius=0)
                Wait Sleep waitTime=0.3
                Set DigitalOutput pin=config_out[1]; digitalValue=1
                Wait Sleep waitTime=0.3
                Loop Counting (count=2) loopVariable(name=Loop_25)
                  bajar := pose_add(get_actual_tcp_pose(), bajada_broca)
                  Waypoint Waypoint (Variable): motionParameters(jointSpeed=1.047198 jointAcceleration=1.396263 cartesianSpeed=0.001 cartesianAcceleration=0.005); variable=bajar
                  subir := pose_sub(get_actual_tcp_pose(), bajada_broca)
                  Waypoint Waypoint (Variable): motionParameters(jointSpeed=1.047198 jointAcceleration=1.396263 cartesianSpeed=0.01 cartesianAcceleration=0.01); variable=subir
                  bajada_broca := pose_sub(bajada_broca, bajada)
                MoveDirectionNode (selectedDirection=ZPlus toolParams=0.03, 0.035)
                  Until DISTANCE (allowActions=false deceleration=3 distanceNodeType=STOP) Distance=0.06; motionParameters(blendRadius=0)
                Set DigitalOutput pin=config_out[1]; digitalValue=0
                barreno_actual := barreno_actual+1
                SuppressedNode
                  Call Quitar_broca
                SuppressedNode
                  Call Poner_broca
        Folder EF
          'desbaste_inicial'
          bajada_broca := p[0,0,-0.012,0,0,0]
          barrenos_menos1 := 8
          barreno_actual := 0
          Loop While (checkContinuously=false) expression=barreno_actual≤barrenos_menos1
            Folder Perforacion
              MoveL speed 100 mm/s, acceleration 500 mm/s^2 (useActiveTCP=true) feature=Base
                internos := interpolate_pose(Linea3_E, Linea3_F, barreno_actual/barrenos_menos1)
                Waypoint Waypoint (Variable): variable=internos
                'desbaste_inicial'
                bajada_broca := p[0,0,-0.012,0,0,0]
                bajada := p[0,0,0.012,0,0,0]
                MoveDirectionNode (selectedDirection=ZMinus toolParams=0.02, 0.015)
                  Until DISTANCE (allowActions=false deceleration=3 distanceNodeType=STOP) Distance=0.055; motionParameters(blendRadius=0)
                Popup Message (haltProgram=false message=punto contacto alanzdo inputType=Text)
                MoveDirectionNode (selectedDirection=ZPlus toolParams=0.003, 0.005)
                  Until DISTANCE (allowActions=false deceleration=3 distanceNodeType=STOP) Distance=0.001; motionParameters(blendRadius=0)
                Wait Sleep waitTime=0.3
                Set DigitalOutput pin=config_out[1]; digitalValue=1
                Wait Sleep waitTime=0.3
                Loop Counting (count=2) loopVariable(name=Loop_27)
                  bajar := pose_add(get_actual_tcp_pose(), bajada_broca)
                  Waypoint Waypoint (Variable): motionParameters(jointSpeed=1.047198 jointAcceleration=1.396263 cartesianSpeed=0.001 cartesianAcceleration=0.005); variable=bajar
                  subir := pose_sub(get_actual_tcp_pose(), bajada_broca)
                  Waypoint Waypoint (Variable): motionParameters(jointSpeed=1.047198 jointAcceleration=1.396263 cartesianSpeed=0.01 cartesianAcceleration=0.01); variable=subir
                  bajada_broca := pose_sub(bajada_broca, bajada)
                MoveDirectionNode (selectedDirection=ZPlus toolParams=0.03, 0.035)
                  Until DISTANCE (allowActions=false deceleration=3 distanceNodeType=STOP) Distance=0.06; motionParameters(blendRadius=0)
                Set DigitalOutput pin=config_out[1]; digitalValue=0
                barreno_actual := barreno_actual+1
                SuppressedNode
                  Call Quitar_broca
                SuppressedNode
                  Call Poner_broca
      Popup Message (haltProgram=false message=Linea3 con media Terminada! inputType=Text)
      Folder Linea4
        Folder Marcar_puntos
          MoveL speed 100 mm/s, acceleration 500 mm/s^2 (useActiveTCP=true) feature=Base
            Waypoint Home3: TCP in base x=-850.182 y=0 z=211.32 mm, rx=-2.0297 ry=2.3968 rz=0.0066 rad; joints [-14.374, -75.698, 98.757, -22.649, -284.037, -0.192] deg; TCP offset x=0.411 y=-218.298 z=37.994 mm, rx=1.558 ry=-0.1255 rz=0.1212 rad
            Waypoint Linea4_A: TCP in base x=-483.35 y=19.133 z=80.413 mm, rx=-2.0297 ry=2.3968 rz=0.0066 rad; joints [-34.857, -105.949, 143.743, -37.281, -304.535, -0.37] deg
            Waypoint Linea4_B: TCP in base x=-685.405 y=19.216 z=80.605 mm, rx=-2.0297 ry=2.3968 rz=0.0066 rad; joints [-21.02, -83.488, 123.782, -39.869, -290.712, -0.217] deg
            Waypoint Linea4_C: TCP in base x=-711.768 y=19.56 z=80.904 mm, rx=-2.0297 ry=2.3968 rz=0.0066 rad; joints [-20.032, -81.151, 120.968, -39.396, -289.723, -0.208] deg
            Waypoint Linea4_D: TCP in base x=-914.58 y=19.801 z=80.703 mm, rx=-2.0297 ry=2.3968 rz=0.0066 rad; joints [-14.612, -64.317, 97.516, -32.795, -284.295, -0.166] deg
            Waypoint Linea4_E: TCP in base x=-939.799 y=20.701 z=80.126 mm, rx=-2.0297 ry=2.3968 rz=0.0066 rad; joints [-14.202, -62.236, 94.311, -31.673, -283.882, -0.163] deg
            Waypoint Linea4_F: TCP in base x=-1143.008 y=20.924 z=80.361 mm, rx=-2.0297 ry=2.3968 rz=0.0066 rad; joints [-11.271, -44.369, 63.742, -18.977, -280.923, -0.147] deg
        Folder AB
          'desbaste_inicial'
          bajada_broca := p[0,0,-0.012,0,0,0]
          barrenos_menos1 := 8
          barreno_actual := 0
          Loop While (checkContinuously=false) expression=barreno_actual≤barrenos_menos1
            Folder Perforacion
              MoveL speed 100 mm/s, acceleration 500 mm/s^2 (useActiveTCP=true) feature=Base
                internos := interpolate_pose(Linea4_A, Linea4_B, barreno_actual/barrenos_menos1)
                Waypoint Waypoint (Variable): variable=internos
                'desbaste_inicial'
                bajada_broca := p[0,0,-0.012,0,0,0]
                bajada := p[0,0,0.012,0,0,0]
                MoveDirectionNode (selectedDirection=ZMinus toolParams=0.02, 0.015)
                  Until DISTANCE (allowActions=false deceleration=3 distanceNodeType=STOP) Distance=0.055; motionParameters(blendRadius=0)
                Popup Message (haltProgram=false message=punto contacto alanzdo inputType=Text)
                MoveDirectionNode (selectedDirection=ZPlus toolParams=0.003, 0.005)
                  Until DISTANCE (allowActions=false deceleration=3 distanceNodeType=STOP) Distance=0.001; motionParameters(blendRadius=0)
                Wait Sleep waitTime=0.3
                Set DigitalOutput pin=config_out[1]; digitalValue=1
                Wait Sleep waitTime=0.3
                Loop Counting (count=2) loopVariable(name=Loop_29)
                  bajar := pose_add(get_actual_tcp_pose(), bajada_broca)
                  Waypoint Waypoint (Variable): motionParameters(jointSpeed=1.047198 jointAcceleration=1.396263 cartesianSpeed=0.001 cartesianAcceleration=0.005); variable=bajar
                  subir := pose_sub(get_actual_tcp_pose(), bajada_broca)
                  Waypoint Waypoint (Variable): motionParameters(jointSpeed=1.047198 jointAcceleration=1.396263 cartesianSpeed=0.01 cartesianAcceleration=0.01); variable=subir
                  bajada_broca := pose_sub(bajada_broca, bajada)
                MoveDirectionNode (selectedDirection=ZPlus toolParams=0.03, 0.035)
                  Until DISTANCE (allowActions=false deceleration=3 distanceNodeType=STOP) Distance=0.06; motionParameters(blendRadius=0)
                Set DigitalOutput pin=config_out[1]; digitalValue=0
                barreno_actual := barreno_actual+1
                SuppressedNode
                  Call Quitar_broca
                SuppressedNode
                  Call Poner_broca
        Folder CD
          'desbaste_inicial'
          bajada_broca := p[0,0,-0.012,0,0,0]
          barrenos_menos1 := 8
          barreno_actual := 0
          Loop While (checkContinuously=false) expression=barreno_actual≤barrenos_menos1
            Folder Perforacion
              MoveL speed 100 mm/s, acceleration 500 mm/s^2 (useActiveTCP=true) feature=Base
                internos := interpolate_pose(Linea4_C, Linea4_D, barreno_actual/barrenos_menos1)
                Waypoint Waypoint (Variable): variable=internos
                'desbaste_inicial'
                bajada_broca := p[0,0,-0.012,0,0,0]
                bajada := p[0,0,0.012,0,0,0]
                MoveDirectionNode (selectedDirection=ZMinus toolParams=0.02, 0.015)
                  Until DISTANCE (allowActions=false deceleration=3 distanceNodeType=STOP) Distance=0.055; motionParameters(blendRadius=0)
                Popup Message (haltProgram=false message=punto contacto alanzdo inputType=Text)
                MoveDirectionNode (selectedDirection=ZPlus toolParams=0.003, 0.005)
                  Until DISTANCE (allowActions=false deceleration=3 distanceNodeType=STOP) Distance=0.001; motionParameters(blendRadius=0)
                Wait Sleep waitTime=0.3
                Set DigitalOutput pin=config_out[1]; digitalValue=1
                Wait Sleep waitTime=0.3
                Loop Counting (count=2) loopVariable(name=Loop_31)
                  bajar := pose_add(get_actual_tcp_pose(), bajada_broca)
                  Waypoint Waypoint (Variable): motionParameters(jointSpeed=1.047198 jointAcceleration=1.396263 cartesianSpeed=0.001 cartesianAcceleration=0.005); variable=bajar
                  subir := pose_sub(get_actual_tcp_pose(), bajada_broca)
                  Waypoint Waypoint (Variable): motionParameters(jointSpeed=1.047198 jointAcceleration=1.396263 cartesianSpeed=0.01 cartesianAcceleration=0.01); variable=subir
                  bajada_broca := pose_sub(bajada_broca, bajada)
                MoveDirectionNode (selectedDirection=ZPlus toolParams=0.03, 0.035)
                  Until DISTANCE (allowActions=false deceleration=3 distanceNodeType=STOP) Distance=0.06; motionParameters(blendRadius=0)
                Set DigitalOutput pin=config_out[1]; digitalValue=0
                barreno_actual := barreno_actual+1
                SuppressedNode
                  Call Quitar_broca
                SuppressedNode
                  Call Poner_broca
        Folder EF
          'desbaste_inicial'
          bajada_broca := p[0,0,-0.012,0,0,0]
          barrenos_menos1 := 8
          barreno_actual := 0
          Loop While (checkContinuously=false) expression=barreno_actual≤barrenos_menos1
            Folder Perforacion
              MoveL speed 100 mm/s, acceleration 500 mm/s^2 (useActiveTCP=true) feature=Base
                internos := interpolate_pose(Linea4_E, Linea4_F, barreno_actual/barrenos_menos1)
                Waypoint Waypoint (Variable): variable=internos
                'desbaste_inicial'
                bajada_broca := p[0,0,-0.012,0,0,0]
                bajada := p[0,0,0.012,0,0,0]
                MoveDirectionNode (selectedDirection=ZMinus toolParams=0.02, 0.015)
                  Until DISTANCE (allowActions=false deceleration=3 distanceNodeType=STOP) Distance=0.055; motionParameters(blendRadius=0)
                Popup Message (haltProgram=false message=punto contacto alanzdo inputType=Text)
                MoveDirectionNode (selectedDirection=ZPlus toolParams=0.003, 0.005)
                  Until DISTANCE (allowActions=false deceleration=3 distanceNodeType=STOP) Distance=0.001; motionParameters(blendRadius=0)
                Wait Sleep waitTime=0.3
                Set DigitalOutput pin=config_out[1]; digitalValue=1
                Wait Sleep waitTime=0.3
                Loop Counting (count=2) loopVariable(name=Loop_33)
                  bajar := pose_add(get_actual_tcp_pose(), bajada_broca)
                  Waypoint Waypoint (Variable): motionParameters(jointSpeed=1.047198 jointAcceleration=1.396263 cartesianSpeed=0.001 cartesianAcceleration=0.005); variable=bajar
                  subir := pose_sub(get_actual_tcp_pose(), bajada_broca)
                  Waypoint Waypoint (Variable): motionParameters(jointSpeed=1.047198 jointAcceleration=1.396263 cartesianSpeed=0.01 cartesianAcceleration=0.01); variable=subir
                  bajada_broca := pose_sub(bajada_broca, bajada)
                MoveDirectionNode (selectedDirection=ZPlus toolParams=0.03, 0.035)
                  Until DISTANCE (allowActions=false deceleration=3 distanceNodeType=STOP) Distance=0.06; motionParameters(blendRadius=0)
                Set DigitalOutput pin=config_out[1]; digitalValue=0
                barreno_actual := barreno_actual+1
                If barreno_actual≥barrenos_menos1
                  cambiar_broca := True
                SuppressedNode
                  Call Quitar_broca
                SuppressedNode
                  Call Poner_broca
      Popup Message (haltProgram=false message=Linea4 con media Terminada! inputType=Text)
    Folder Broca_3
      Folder Linea3
        Folder Marcar_puntos
          MoveL speed 100 mm/s, acceleration 500 mm/s^2 (useActiveTCP=true) feature=Base
            Waypoint Home3: TCP in base x=-850.182 y=0 z=211.32 mm, rx=-2.0297 ry=2.3968 rz=0.0066 rad; joints [-14.374, -75.698, 98.757, -22.649, -284.037, -0.192] deg
            Waypoint Linea3_A: TCP in base x=-483.981 y=-387.033 z=81.05 mm, rx=-2.0297 ry=2.3968 rz=0.0065 rad; joints [29.472, -85.66, 126.185, -40.12, -240.222, 0.138] deg; TCP offset x=0.411 y=-218.298 z=37.994 mm, rx=1.558 ry=-0.1255 rz=0.1212 rad
            Waypoint Linea3_B: TCP in base x=-686.975 y=-386.566 z=81.205 mm, rx=-2.0297 ry=2.3968 rz=0.0065 rad; joints [20.619, -72.662, 109.808, -36.76, -249.072, 0.076] deg
            Waypoint Linea3_C: TCP in base x=-712.354 y=-386.033 z=80.584 mm, rx=-2.0297 ry=2.3968 rz=0.0065 rad; joints [19.8, -70.954, 107.463, -36.125, -249.889, 0.07] deg
            Waypoint Linea3_D: TCP in base x=-915.146 y=-385.55 z=81.731 mm, rx=-2.0297 ry=2.3968 rz=0.0065 rad; joints [15.111, -56.737, 85.163, -28.047, -254.563, 0.035] deg
            Waypoint Linea3_E: TCP in base x=-940.448 y=-385.682 z=81.142 mm, rx=-2.0297 ry=2.3968 rz=0.0065 rad; joints [14.681, -54.779, 81.937, -26.78, -254.99, 0.031] deg
            Waypoint Linea3_F: TCP in base x=-1144.267 y=-385.383 z=81.233 mm, rx=-2.0297 ry=2.3968 rz=0.0065 rad; joints [11.857, -36.303, 48.734, -12.056, -257.778, 0.006] deg
        Folder AB
          'desbaste_inicial'
          bajada_broca := p[0,0,-0.024,0,0,0]
          barrenos_menos1 := 8
          barreno_actual := 0
          Loop While (checkContinuously=false) expression=barreno_actual≤barrenos_menos1
            Folder Perforacion
              MoveL speed 100 mm/s, acceleration 500 mm/s^2 (useActiveTCP=true) feature=Base
                internos := interpolate_pose(Linea3_A, Linea3_B, barreno_actual/barrenos_menos1)
                Waypoint Waypoint (Variable): variable=internos
                'desbaste_inicial'
                bajada_broca := p[0,0,-0.024,0,0,0]
                bajada := p[0,0,0.024,0,0,0]
                MoveDirectionNode (selectedDirection=ZMinus toolParams=0.02, 0.015)
                  Until DISTANCE (allowActions=false deceleration=3 distanceNodeType=STOP) Distance=0.055; motionParameters(blendRadius=0)
                Popup Message (haltProgram=false message=punto contacto alanzdo inputType=Text)
                MoveDirectionNode (selectedDirection=ZPlus toolParams=0.003, 0.005)
                  Until DISTANCE (allowActions=false deceleration=3 distanceNodeType=STOP) Distance=0.001; motionParameters(blendRadius=0)
                Wait Sleep waitTime=0.3
                Set DigitalOutput pin=config_out[1]; digitalValue=1
                Wait Sleep waitTime=0.3
                Loop Counting (count=1) loopVariable(name=Loop_37)
                  bajar := pose_add(get_actual_tcp_pose(), bajada_broca)
                  Waypoint Waypoint (Variable): motionParameters(jointSpeed=1.047198 jointAcceleration=1.396263 cartesianSpeed=0.001 cartesianAcceleration=0.005); variable=bajar
                  subir := pose_sub(get_actual_tcp_pose(), bajada_broca)
                  Waypoint Waypoint (Variable): motionParameters(jointSpeed=1.047198 jointAcceleration=1.396263 cartesianSpeed=0.01 cartesianAcceleration=0.01); variable=subir
                  bajada_broca := pose_sub(bajada_broca, bajada)
                MoveDirectionNode (selectedDirection=ZPlus toolParams=0.03, 0.035)
                  Until DISTANCE (allowActions=false deceleration=3 distanceNodeType=STOP) Distance=0.06; motionParameters(blendRadius=0)
                Set DigitalOutput pin=config_out[1]; digitalValue=0
                barreno_actual := barreno_actual+1
                SuppressedNode
                  Call Quitar_broca
                SuppressedNode
                  Call Poner_broca
        Folder CD
          'desbaste_inicial'
          bajada_broca := p[0,0,-0.024,0,0,0]
          barrenos_menos1 := 8
          barreno_actual := 0
          Loop While (checkContinuously=false) expression=barreno_actual≤barrenos_menos1
            Folder Perforacion
              MoveL speed 100 mm/s, acceleration 500 mm/s^2 (useActiveTCP=true) feature=Base
                internos := interpolate_pose(Linea3_C, Linea3_D, barreno_actual/barrenos_menos1)
                Waypoint Waypoint (Variable): variable=internos
                'desbaste_inicial'
                bajada_broca := p[0,0,-0.024,0,0,0]
                bajada := p[0,0,0.024,0,0,0]
                MoveDirectionNode (selectedDirection=ZMinus toolParams=0.02, 0.015)
                  Until DISTANCE (allowActions=false deceleration=3 distanceNodeType=STOP) Distance=0.055; motionParameters(blendRadius=0)
                Popup Message (haltProgram=false message=punto contacto alanzdo inputType=Text)
                MoveDirectionNode (selectedDirection=ZPlus toolParams=0.003, 0.005)
                  Until DISTANCE (allowActions=false deceleration=3 distanceNodeType=STOP) Distance=0.001; motionParameters(blendRadius=0)
                Wait Sleep waitTime=0.3
                Set DigitalOutput pin=config_out[1]; digitalValue=1
                Wait Sleep waitTime=0.3
                Loop Counting (count=1) loopVariable(name=Loop_41)
                  bajar := pose_add(get_actual_tcp_pose(), bajada_broca)
                  Waypoint Waypoint (Variable): motionParameters(jointSpeed=1.047198 jointAcceleration=1.396263 cartesianSpeed=0.001 cartesianAcceleration=0.005); variable=bajar
                  subir := pose_sub(get_actual_tcp_pose(), bajada_broca)
                  Waypoint Waypoint (Variable): motionParameters(jointSpeed=1.047198 jointAcceleration=1.396263 cartesianSpeed=0.01 cartesianAcceleration=0.01); variable=subir
                  bajada_broca := pose_sub(bajada_broca, bajada)
                MoveDirectionNode (selectedDirection=ZPlus toolParams=0.03, 0.035)
                  Until DISTANCE (allowActions=false deceleration=3 distanceNodeType=STOP) Distance=0.06; motionParameters(blendRadius=0)
                Set DigitalOutput pin=config_out[1]; digitalValue=0
                barreno_actual := barreno_actual+1
                SuppressedNode
                  Call Quitar_broca
                SuppressedNode
                  Call Poner_broca
        Folder EF
          'desbaste_inicial'
          bajada_broca := p[0,0,-0.024,0,0,0]
          barrenos_menos1 := 8
          barreno_actual := 0
          Loop While (checkContinuously=false) expression=barreno_actual≤barrenos_menos1
            Folder Perforacion
              MoveL speed 100 mm/s, acceleration 500 mm/s^2 (useActiveTCP=true) feature=Base
                internos := interpolate_pose(Linea3_E, Linea3_F, barreno_actual/barrenos_menos1)
                Waypoint Waypoint (Variable): variable=internos
                'desbaste_inicial'
                bajada_broca := p[0,0,-0.024,0,0,0]
                bajada := p[0,0,0.024,0,0,0]
                MoveDirectionNode (selectedDirection=ZMinus toolParams=0.02, 0.015)
                  Until DISTANCE (allowActions=false deceleration=3 distanceNodeType=STOP) Distance=0.055; motionParameters(blendRadius=0)
                Popup Message (haltProgram=false message=punto contacto alanzdo inputType=Text)
                MoveDirectionNode (selectedDirection=ZPlus toolParams=0.003, 0.005)
                  Until DISTANCE (allowActions=false deceleration=3 distanceNodeType=STOP) Distance=0.001; motionParameters(blendRadius=0)
                Wait Sleep waitTime=0.3
                Set DigitalOutput pin=config_out[1]; digitalValue=1
                Wait Sleep waitTime=0.3
                Loop Counting (count=1) loopVariable(name=Loop_45)
                  bajar := pose_add(get_actual_tcp_pose(), bajada_broca)
                  Waypoint Waypoint (Variable): motionParameters(jointSpeed=1.047198 jointAcceleration=1.396263 cartesianSpeed=0.001 cartesianAcceleration=0.005); variable=bajar
                  subir := pose_sub(get_actual_tcp_pose(), bajada_broca)
                  Waypoint Waypoint (Variable): motionParameters(jointSpeed=1.047198 jointAcceleration=1.396263 cartesianSpeed=0.01 cartesianAcceleration=0.01); variable=subir
                  bajada_broca := pose_sub(bajada_broca, bajada)
                MoveDirectionNode (selectedDirection=ZPlus toolParams=0.03, 0.035)
                  Until DISTANCE (allowActions=false deceleration=3 distanceNodeType=STOP) Distance=0.06; motionParameters(blendRadius=0)
                Set DigitalOutput pin=config_out[1]; digitalValue=0
                barreno_actual := barreno_actual+1
                SuppressedNode
                  Call Quitar_broca
                SuppressedNode
                  Call Poner_broca
      Popup Message (haltProgram=false message=Linea3 con full Terminada! inputType=Text)
      Folder Linea4
        Folder Marcar_puntos
          MoveL speed 100 mm/s, acceleration 500 mm/s^2 (useActiveTCP=true) feature=Base
            Waypoint Home3: TCP in base x=-850.182 y=0 z=211.32 mm, rx=-2.0297 ry=2.3968 rz=0.0066 rad; joints [-14.374, -75.698, 98.757, -22.649, -284.037, -0.192] deg; TCP offset x=0.411 y=-218.298 z=37.994 mm, rx=1.558 ry=-0.1255 rz=0.1212 rad
            Waypoint Linea4_A: TCP in base x=-483.35 y=19.133 z=80.413 mm, rx=-2.0297 ry=2.3968 rz=0.0066 rad; joints [-34.857, -105.949, 143.743, -37.281, -304.535, -0.37] deg
            Waypoint Linea4_B: TCP in base x=-685.405 y=19.216 z=80.605 mm, rx=-2.0297 ry=2.3968 rz=0.0066 rad; joints [-21.02, -83.488, 123.782, -39.869, -290.712, -0.217] deg
            Waypoint Linea4_C: TCP in base x=-711.768 y=19.56 z=80.904 mm, rx=-2.0297 ry=2.3968 rz=0.0066 rad; joints [-20.032, -81.151, 120.968, -39.396, -289.723, -0.208] deg
            Waypoint Linea4_D: TCP in base x=-914.58 y=19.801 z=80.703 mm, rx=-2.0297 ry=2.3968 rz=0.0066 rad; joints [-14.612, -64.317, 97.516, -32.795, -284.295, -0.166] deg
            Waypoint Linea4_E: TCP in base x=-939.799 y=20.701 z=80.126 mm, rx=-2.0297 ry=2.3968 rz=0.0066 rad; joints [-14.202, -62.236, 94.311, -31.673, -283.882, -0.163] deg
            Waypoint Linea4_F: TCP in base x=-1143.008 y=20.924 z=80.361 mm, rx=-2.0297 ry=2.3968 rz=0.0066 rad; joints [-11.271, -44.369, 63.742, -18.977, -280.923, -0.147] deg
        Folder AB
          'desbaste_inicial'
          bajada_broca := p[0,0,-0.024,0,0,0]
          barrenos_menos1 := 8
          barreno_actual := 0
